// TIA Portal V16 export
// export: Created 2023-06-21T17:06:21.6795389Z, ExportSetting WithDefaults, DisplayName Totally Integrated Automation Portal, DisplayVersion V16 Update 4, DisplayName TIA Portal Version Control Interface, DisplayVersion V16 Update 2, DisplayName TIA Portal Openness, DisplayVersion V16 Update 4, DisplayName SINAMICS Startdrive Advanced, DisplayVersion V16, DisplayName SINAMICS Startdrive G130, G150, S120, S150, SINAMICS MV, S210, DisplayVersion V16, DisplayName SINAMICS Startdrive G110M, G120, G120C, G120D, G120P, DisplayVersion V16, DisplayName STEP 7 Professional, DisplayVersion V16 Update 4, DisplayName STEP 7 Safety, DisplayVersion V16, DisplayName Soft Starter ES, DisplayVersion V16, DisplayName WinCC Advanced, DisplayVersion V16 Update 4
ORGANIZATION_BLOCK "Cyclic interrupt"   // OB30, LAD, CyclicInterrupt
{ S7_Optimized_Access := 'TRUE' }
VERSION : 0.1
// stored: AutoNumber true, IsIECCheckEnabled false, SetENOAutomatically false
   VAR_INPUT
      Initial_Call : Bool;   // Initial call of this OB
      Event_Count : Int;   // Events discarded
   END_VAR
   VAR_TEMP
      Aux_SP_1 : Int;
      Aux_SP_2 : Int;
      Aux_SP_3 : Int;
      Aux_SP_4 : Int;
      Aux_SP_5 : Int;
      Aux_SP_6 : Int;
      Aux_SP_7 : Int;
      Aux_SP_8 : Int;
      Aux_SP_9 : Int;
      Aux_SP_10 : Int;
      Aux_SP_11 : Int;
      Aux_SP_12 : Int;
      Aux_SP_13 : Int;
      Aux_SP_14 : Int;
   END_VAR
   VAR_TEMP   // added for the SCL form of the ladder/FBD networks
      _w1 : Bool;
   END_VAR
BEGIN

REGION Network 2: START
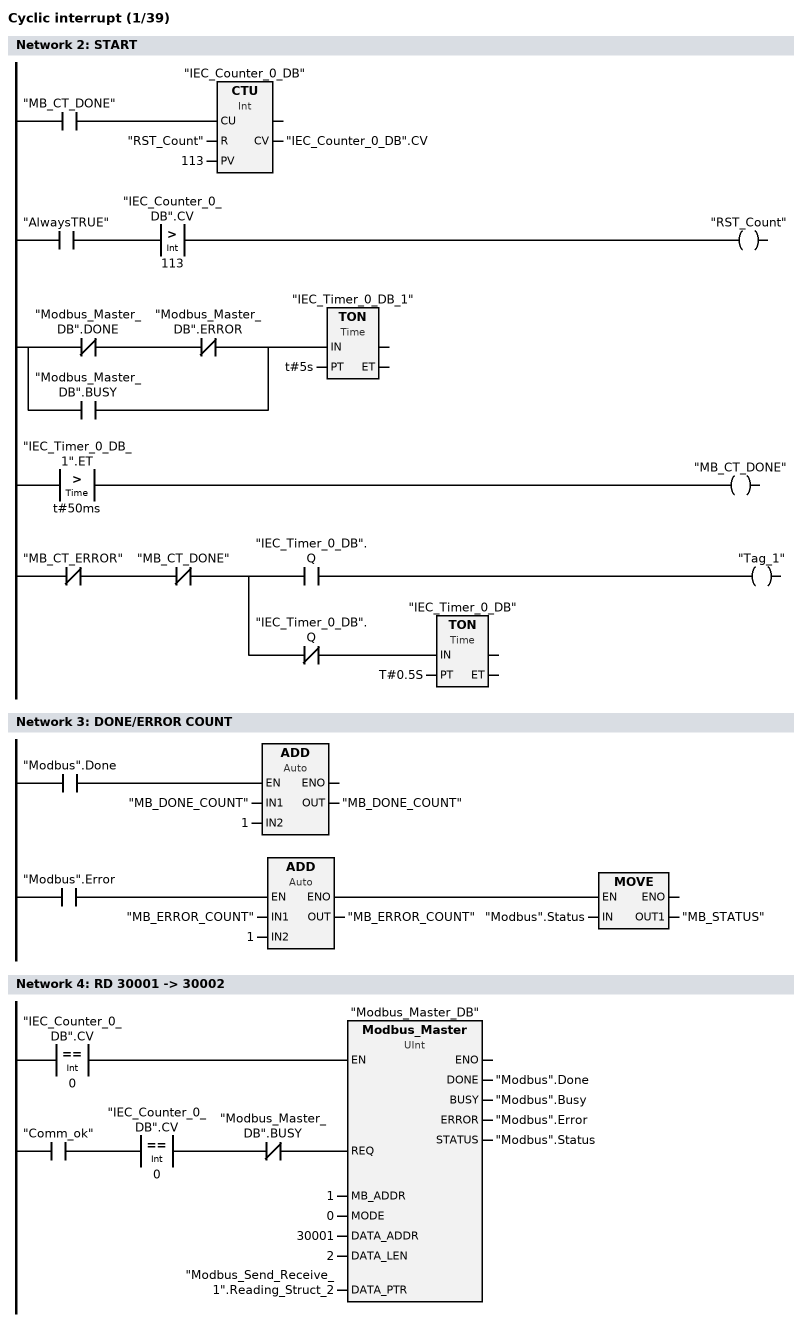
   RUNG wire#powerrail
      Contact( "MB_CT_DONE" )
      { S7_Templates := "value_type := Int" } "IEC_Counter_0_DB".CTU(r := "RST_Count", pv := 113, cv => "IEC_Counter_0_DB".CV)
   END_RUNG
   RUNG wire#powerrail
      Contact( "AlwaysTRUE" )
      { S7_Templates := "SrcType := Int" } GT_Contact(in1 := "IEC_Counter_0_DB".CV, in2 := 113)
      Coil( "RST_Count" )
   END_RUNG
   RUNG wire#powerrail
      I_Contact( "Modbus_Master_DB".DONE )
      I_Contact( "Modbus_Master_DB".ERROR )
      wire#w1
      { S7_Templates := "time_type := Time" } "IEC_Timer_0_DB_1".TON(pt := t#5s, et =>)
   END_RUNG
   RUNG wire#powerrail
      Contact( "Modbus_Master_DB".BUSY )
   END_RUNG wire#w1
   RUNG wire#powerrail
      { S7_Templates := "SrcType := Time" } GT_Contact(in1 := "IEC_Timer_0_DB_1".ET, in2 := t#50ms)
      Coil( "MB_CT_DONE" )
   END_RUNG
   RUNG wire#powerrail
      I_Contact( "MB_CT_ERROR" )
      I_Contact( "MB_CT_DONE" )
      wire#w2
      Contact( "IEC_Timer_0_DB".Q )
      Coil( "Tag_1" )
   END_RUNG
   RUNG wire#w2
      I_Contact( "IEC_Timer_0_DB".Q )
      { S7_Templates := "time_type := Time" } "IEC_Timer_0_DB".TON(pt := T#0.5S, et =>)
   END_RUNG
   // the same network as SCL:
   "IEC_Counter_0_DB".CTU(CU := "MB_CT_DONE", R := "RST_Count", PV := 113, CV => "IEC_Counter_0_DB".CV);
   "RST_Count" := "AlwaysTRUE" AND ("IEC_Counter_0_DB".CV > 113);
   "IEC_Timer_0_DB_1".TON(IN := (NOT "Modbus_Master_DB".DONE AND NOT "Modbus_Master_DB".ERROR) OR "Modbus_Master_DB".BUSY,
                          PT := t#5s);
   "MB_CT_DONE" := "IEC_Timer_0_DB_1".ET > t#50ms;
   #_w1 := NOT "MB_CT_ERROR" AND NOT "MB_CT_DONE";
   "Tag_1" := #_w1 AND "IEC_Timer_0_DB".Q;
   "IEC_Timer_0_DB".TON(IN := #_w1 AND NOT "IEC_Timer_0_DB".Q, PT := T#0.5S);
END_REGION

REGION Network 3: DONE/ERROR COUNT
   RUNG wire#powerrail
      Contact( "Modbus".Done )
      Add(in1 := "MB_DONE_COUNT", in2 := 1, out => "MB_DONE_COUNT")
   END_RUNG
   RUNG wire#powerrail
      Contact( "Modbus".Error )
      Add(in1 := "MB_ERROR_COUNT", in2 := 1, out => "MB_ERROR_COUNT")
      Move(in := "Modbus".Status, out1 => "MB_STATUS")
   END_RUNG
   // the same network as SCL:
   IF "Modbus".Done THEN "MB_DONE_COUNT" := "MB_DONE_COUNT" + 1; END_IF;
   IF "Modbus".Error THEN
       "MB_ERROR_COUNT" := "MB_ERROR_COUNT" + 1;
       "MB_STATUS" := "Modbus".Status;
   END_IF;
END_REGION

REGION Network 4: RD 30001 -> 30002
   RUNG wire#powerrail
      { S7_Templates := "SrcType := Int" } EQ_Contact(in1 := "IEC_Counter_0_DB".CV, in2 := 0)
      { S7_Templates := "[card := 0, word_type := UInt, dword_type := UDInt, byte_type := USInt, any_type := Variant]" } "Modbus_Master_DB".Modbus_Master(REQ := wire#w1, MB_ADDR := 1, MODE := 0, DATA_ADDR := 30001, DATA_LEN := 2, DATA_PTR := "Modbus_Send_Receive_1".Reading_Struct_2, DONE => "Modbus".Done, BUSY => "Modbus".Busy, ERROR => "Modbus".Error, STATUS => "Modbus".Status)
   END_RUNG
   RUNG wire#powerrail
      Contact( "Comm_ok" )
      { S7_Templates := "SrcType := Int" } EQ_Contact(in1 := "IEC_Counter_0_DB".CV, in2 := 0)
      I_Contact( "Modbus_Master_DB".BUSY )
   END_RUNG wire#w1
   // the same network as SCL:
   IF "IEC_Counter_0_DB".CV = 0 THEN
       "Modbus_Master_DB"(REQ := "Comm_ok" AND ("IEC_Counter_0_DB".CV = 0) AND NOT "Modbus_Master_DB".BUSY,   // Modbus_Master
                          MB_ADDR := 1,
                          MODE := 0,
                          DATA_ADDR := 30001,
                          DATA_LEN := 2,
                          DATA_PTR := "Modbus_Send_Receive_1".Reading_Struct_2,
                          DONE => "Modbus".Done,
                          BUSY => "Modbus".Busy,
                          ERROR => "Modbus".Error,
                          STATUS => "Modbus".Status);
   END_IF;
END_REGION

REGION Network 5: STS MAN/AUTO
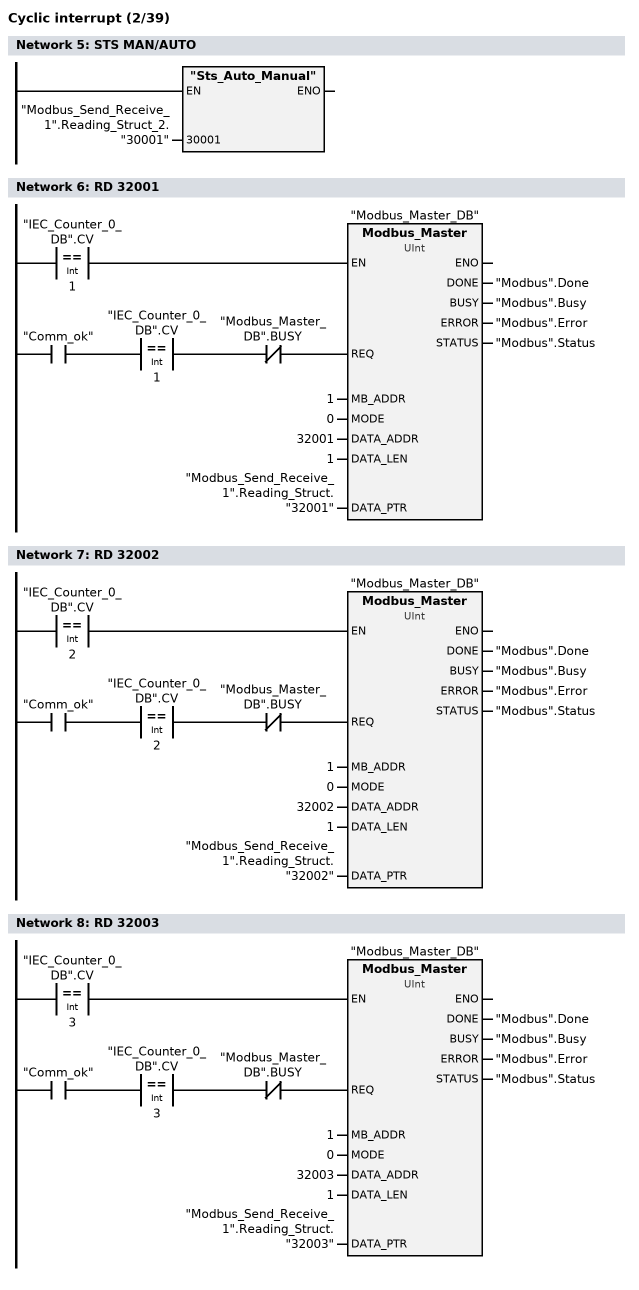
   RUNG wire#powerrail
      "Sts_Auto_Manual"("30001" := "Modbus_Send_Receive_1".Reading_Struct_2."30001")
   END_RUNG
   // the same network as SCL:
   "Sts_Auto_Manual"("30001" := "Modbus_Send_Receive_1".Reading_Struct_2."30001");
END_REGION

REGION Network 6: RD 32001
   RUNG wire#powerrail
      { S7_Templates := "SrcType := Int" } EQ_Contact(in1 := "IEC_Counter_0_DB".CV, in2 := 1)
      { S7_Templates := "[card := 0, word_type := UInt, dword_type := UDInt, byte_type := USInt, any_type := Variant]" } "Modbus_Master_DB".Modbus_Master(REQ := wire#w1, MB_ADDR := 1, MODE := 0, DATA_ADDR := 32001, DATA_LEN := 1, DATA_PTR := "Modbus_Send_Receive_1".Reading_Struct."32001", DONE => "Modbus".Done, BUSY => "Modbus".Busy, ERROR => "Modbus".Error, STATUS => "Modbus".Status)
   END_RUNG
   RUNG wire#powerrail
      Contact( "Comm_ok" )
      { S7_Templates := "SrcType := Int" } EQ_Contact(in1 := "IEC_Counter_0_DB".CV, in2 := 1)
      I_Contact( "Modbus_Master_DB".BUSY )
   END_RUNG wire#w1
   // the same network as SCL:
   IF "IEC_Counter_0_DB".CV = 1 THEN
       "Modbus_Master_DB"(REQ := "Comm_ok" AND ("IEC_Counter_0_DB".CV = 1) AND NOT "Modbus_Master_DB".BUSY,   // Modbus_Master
                          MB_ADDR := 1,
                          MODE := 0,
                          DATA_ADDR := 32001,
                          DATA_LEN := 1,
                          DATA_PTR := "Modbus_Send_Receive_1".Reading_Struct."32001",
                          DONE => "Modbus".Done,
                          BUSY => "Modbus".Busy,
                          ERROR => "Modbus".Error,
                          STATUS => "Modbus".Status);
   END_IF;
END_REGION

REGION Network 7: RD 32002
   RUNG wire#powerrail
      { S7_Templates := "SrcType := Int" } EQ_Contact(in1 := "IEC_Counter_0_DB".CV, in2 := 2)
      { S7_Templates := "[card := 0, word_type := UInt, dword_type := UDInt, byte_type := USInt, any_type := Variant]" } "Modbus_Master_DB".Modbus_Master(REQ := wire#w1, MB_ADDR := 1, MODE := 0, DATA_ADDR := 32002, DATA_LEN := 1, DATA_PTR := "Modbus_Send_Receive_1".Reading_Struct."32002", DONE => "Modbus".Done, BUSY => "Modbus".Busy, ERROR => "Modbus".Error, STATUS => "Modbus".Status)
   END_RUNG
   RUNG wire#powerrail
      Contact( "Comm_ok" )
      { S7_Templates := "SrcType := Int" } EQ_Contact(in1 := "IEC_Counter_0_DB".CV, in2 := 2)
      I_Contact( "Modbus_Master_DB".BUSY )
   END_RUNG wire#w1
   // the same network as SCL:
   IF "IEC_Counter_0_DB".CV = 2 THEN
       "Modbus_Master_DB"(REQ := "Comm_ok" AND ("IEC_Counter_0_DB".CV = 2) AND NOT "Modbus_Master_DB".BUSY,   // Modbus_Master
                          MB_ADDR := 1,
                          MODE := 0,
                          DATA_ADDR := 32002,
                          DATA_LEN := 1,
                          DATA_PTR := "Modbus_Send_Receive_1".Reading_Struct."32002",
                          DONE => "Modbus".Done,
                          BUSY => "Modbus".Busy,
                          ERROR => "Modbus".Error,
                          STATUS => "Modbus".Status);
   END_IF;
END_REGION

REGION Network 8: RD 32003
   RUNG wire#powerrail
      { S7_Templates := "SrcType := Int" } EQ_Contact(in1 := "IEC_Counter_0_DB".CV, in2 := 3)
      { S7_Templates := "[card := 0, word_type := UInt, dword_type := UDInt, byte_type := USInt, any_type := Variant]" } "Modbus_Master_DB".Modbus_Master(REQ := wire#w1, MB_ADDR := 1, MODE := 0, DATA_ADDR := 32003, DATA_LEN := 1, DATA_PTR := "Modbus_Send_Receive_1".Reading_Struct."32003", DONE => "Modbus".Done, BUSY => "Modbus".Busy, ERROR => "Modbus".Error, STATUS => "Modbus".Status)
   END_RUNG
   RUNG wire#powerrail
      Contact( "Comm_ok" )
      { S7_Templates := "SrcType := Int" } EQ_Contact(in1 := "IEC_Counter_0_DB".CV, in2 := 3)
      I_Contact( "Modbus_Master_DB".BUSY )
   END_RUNG wire#w1
   // the same network as SCL:
   IF "IEC_Counter_0_DB".CV = 3 THEN
       "Modbus_Master_DB"(REQ := "Comm_ok" AND ("IEC_Counter_0_DB".CV = 3) AND NOT "Modbus_Master_DB".BUSY,   // Modbus_Master
                          MB_ADDR := 1,
                          MODE := 0,
                          DATA_ADDR := 32003,
                          DATA_LEN := 1,
                          DATA_PTR := "Modbus_Send_Receive_1".Reading_Struct."32003",
                          DONE => "Modbus".Done,
                          BUSY => "Modbus".Busy,
                          ERROR => "Modbus".Error,
                          STATUS => "Modbus".Status);
   END_IF;
END_REGION

REGION Network 9: RD 32004
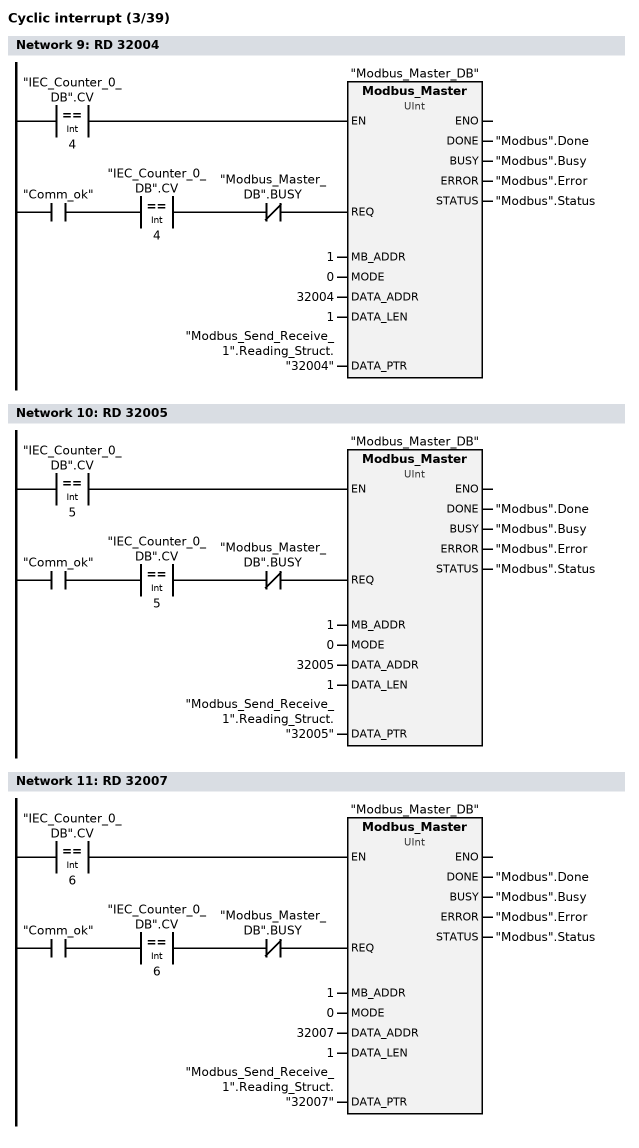
   RUNG wire#powerrail
      { S7_Templates := "SrcType := Int" } EQ_Contact(in1 := "IEC_Counter_0_DB".CV, in2 := 4)
      { S7_Templates := "[card := 0, word_type := UInt, dword_type := UDInt, byte_type := USInt, any_type := Variant]" } "Modbus_Master_DB".Modbus_Master(REQ := wire#w1, MB_ADDR := 1, MODE := 0, DATA_ADDR := 32004, DATA_LEN := 1, DATA_PTR := "Modbus_Send_Receive_1".Reading_Struct."32004", DONE => "Modbus".Done, BUSY => "Modbus".Busy, ERROR => "Modbus".Error, STATUS => "Modbus".Status)
   END_RUNG
   RUNG wire#powerrail
      Contact( "Comm_ok" )
      { S7_Templates := "SrcType := Int" } EQ_Contact(in1 := "IEC_Counter_0_DB".CV, in2 := 4)
      I_Contact( "Modbus_Master_DB".BUSY )
   END_RUNG wire#w1
   // the same network as SCL:
   IF "IEC_Counter_0_DB".CV = 4 THEN
       "Modbus_Master_DB"(REQ := "Comm_ok" AND ("IEC_Counter_0_DB".CV = 4) AND NOT "Modbus_Master_DB".BUSY,   // Modbus_Master
                          MB_ADDR := 1,
                          MODE := 0,
                          DATA_ADDR := 32004,
                          DATA_LEN := 1,
                          DATA_PTR := "Modbus_Send_Receive_1".Reading_Struct."32004",
                          DONE => "Modbus".Done,
                          BUSY => "Modbus".Busy,
                          ERROR => "Modbus".Error,
                          STATUS => "Modbus".Status);
   END_IF;
END_REGION

REGION Network 10: RD 32005
   RUNG wire#powerrail
      { S7_Templates := "SrcType := Int" } EQ_Contact(in1 := "IEC_Counter_0_DB".CV, in2 := 5)
      { S7_Templates := "[card := 0, word_type := UInt, dword_type := UDInt, byte_type := USInt, any_type := Variant]" } "Modbus_Master_DB".Modbus_Master(REQ := wire#w1, MB_ADDR := 1, MODE := 0, DATA_ADDR := 32005, DATA_LEN := 1, DATA_PTR := "Modbus_Send_Receive_1".Reading_Struct."32005", DONE => "Modbus".Done, BUSY => "Modbus".Busy, ERROR => "Modbus".Error, STATUS => "Modbus".Status)
   END_RUNG
   RUNG wire#powerrail
      Contact( "Comm_ok" )
      { S7_Templates := "SrcType := Int" } EQ_Contact(in1 := "IEC_Counter_0_DB".CV, in2 := 5)
      I_Contact( "Modbus_Master_DB".BUSY )
   END_RUNG wire#w1
   // the same network as SCL:
   IF "IEC_Counter_0_DB".CV = 5 THEN
       "Modbus_Master_DB"(REQ := "Comm_ok" AND ("IEC_Counter_0_DB".CV = 5) AND NOT "Modbus_Master_DB".BUSY,   // Modbus_Master
                          MB_ADDR := 1,
                          MODE := 0,
                          DATA_ADDR := 32005,
                          DATA_LEN := 1,
                          DATA_PTR := "Modbus_Send_Receive_1".Reading_Struct."32005",
                          DONE => "Modbus".Done,
                          BUSY => "Modbus".Busy,
                          ERROR => "Modbus".Error,
                          STATUS => "Modbus".Status);
   END_IF;
END_REGION

REGION Network 11: RD 32007
   RUNG wire#powerrail
      { S7_Templates := "SrcType := Int" } EQ_Contact(in1 := "IEC_Counter_0_DB".CV, in2 := 6)
      { S7_Templates := "[card := 0, word_type := UInt, dword_type := UDInt, byte_type := USInt, any_type := Variant]" } "Modbus_Master_DB".Modbus_Master(REQ := wire#w1, MB_ADDR := 1, MODE := 0, DATA_ADDR := 32007, DATA_LEN := 1, DATA_PTR := "Modbus_Send_Receive_1".Reading_Struct."32007", DONE => "Modbus".Done, BUSY => "Modbus".Busy, ERROR => "Modbus".Error, STATUS => "Modbus".Status)
   END_RUNG
   RUNG wire#powerrail
      Contact( "Comm_ok" )
      { S7_Templates := "SrcType := Int" } EQ_Contact(in1 := "IEC_Counter_0_DB".CV, in2 := 6)
      I_Contact( "Modbus_Master_DB".BUSY )
   END_RUNG wire#w1
   // the same network as SCL:
   IF "IEC_Counter_0_DB".CV = 6 THEN
       "Modbus_Master_DB"(REQ := "Comm_ok" AND ("IEC_Counter_0_DB".CV = 6) AND NOT "Modbus_Master_DB".BUSY,   // Modbus_Master
                          MB_ADDR := 1,
                          MODE := 0,
                          DATA_ADDR := 32007,
                          DATA_LEN := 1,
                          DATA_PTR := "Modbus_Send_Receive_1".Reading_Struct."32007",
                          DONE => "Modbus".Done,
                          BUSY => "Modbus".Busy,
                          ERROR => "Modbus".Error,
                          STATUS => "Modbus".Status);
   END_IF;
END_REGION

REGION Network 12: RD 32008
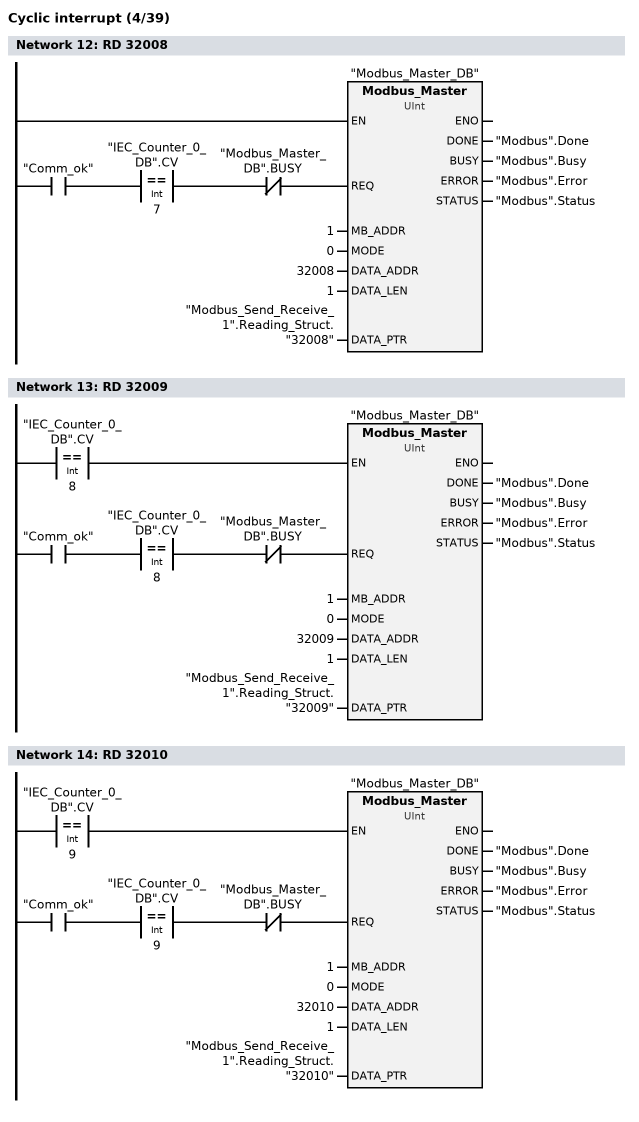
   RUNG wire#powerrail
      { S7_Templates := "[card := 0, word_type := UInt, dword_type := UDInt, byte_type := USInt, any_type := Variant]" } "Modbus_Master_DB".Modbus_Master(REQ := wire#w1, MB_ADDR := 1, MODE := 0, DATA_ADDR := 32008, DATA_LEN := 1, DATA_PTR := "Modbus_Send_Receive_1".Reading_Struct."32008", DONE => "Modbus".Done, BUSY => "Modbus".Busy, ERROR => "Modbus".Error, STATUS => "Modbus".Status)
   END_RUNG
   RUNG wire#powerrail
      Contact( "Comm_ok" )
      { S7_Templates := "SrcType := Int" } EQ_Contact(in1 := "IEC_Counter_0_DB".CV, in2 := 7)
      I_Contact( "Modbus_Master_DB".BUSY )
   END_RUNG wire#w1
   // the same network as SCL:
   "Modbus_Master_DB"(REQ := "Comm_ok" AND ("IEC_Counter_0_DB".CV = 7) AND NOT "Modbus_Master_DB".BUSY,   // Modbus_Master
                      MB_ADDR := 1,
                      MODE := 0,
                      DATA_ADDR := 32008,
                      DATA_LEN := 1,
                      DATA_PTR := "Modbus_Send_Receive_1".Reading_Struct."32008",
                      DONE => "Modbus".Done,
                      BUSY => "Modbus".Busy,
                      ERROR => "Modbus".Error,
                      STATUS => "Modbus".Status);
END_REGION

REGION Network 13: RD 32009
   RUNG wire#powerrail
      { S7_Templates := "SrcType := Int" } EQ_Contact(in1 := "IEC_Counter_0_DB".CV, in2 := 8)
      { S7_Templates := "[card := 0, word_type := UInt, dword_type := UDInt, byte_type := USInt, any_type := Variant]" } "Modbus_Master_DB".Modbus_Master(REQ := wire#w1, MB_ADDR := 1, MODE := 0, DATA_ADDR := 32009, DATA_LEN := 1, DATA_PTR := "Modbus_Send_Receive_1".Reading_Struct."32009", DONE => "Modbus".Done, BUSY => "Modbus".Busy, ERROR => "Modbus".Error, STATUS => "Modbus".Status)
   END_RUNG
   RUNG wire#powerrail
      Contact( "Comm_ok" )
      { S7_Templates := "SrcType := Int" } EQ_Contact(in1 := "IEC_Counter_0_DB".CV, in2 := 8)
      I_Contact( "Modbus_Master_DB".BUSY )
   END_RUNG wire#w1
   // the same network as SCL:
   IF "IEC_Counter_0_DB".CV = 8 THEN
       "Modbus_Master_DB"(REQ := "Comm_ok" AND ("IEC_Counter_0_DB".CV = 8) AND NOT "Modbus_Master_DB".BUSY,   // Modbus_Master
                          MB_ADDR := 1,
                          MODE := 0,
                          DATA_ADDR := 32009,
                          DATA_LEN := 1,
                          DATA_PTR := "Modbus_Send_Receive_1".Reading_Struct."32009",
                          DONE => "Modbus".Done,
                          BUSY => "Modbus".Busy,
                          ERROR => "Modbus".Error,
                          STATUS => "Modbus".Status);
   END_IF;
END_REGION

REGION Network 14: RD 32010
   RUNG wire#powerrail
      { S7_Templates := "SrcType := Int" } EQ_Contact(in1 := "IEC_Counter_0_DB".CV, in2 := 9)
      { S7_Templates := "[card := 0, word_type := UInt, dword_type := UDInt, byte_type := USInt, any_type := Variant]" } "Modbus_Master_DB".Modbus_Master(REQ := wire#w1, MB_ADDR := 1, MODE := 0, DATA_ADDR := 32010, DATA_LEN := 1, DATA_PTR := "Modbus_Send_Receive_1".Reading_Struct."32010", DONE => "Modbus".Done, BUSY => "Modbus".Busy, ERROR => "Modbus".Error, STATUS => "Modbus".Status)
   END_RUNG
   RUNG wire#powerrail
      Contact( "Comm_ok" )
      { S7_Templates := "SrcType := Int" } EQ_Contact(in1 := "IEC_Counter_0_DB".CV, in2 := 9)
      I_Contact( "Modbus_Master_DB".BUSY )
   END_RUNG wire#w1
   // the same network as SCL:
   IF "IEC_Counter_0_DB".CV = 9 THEN
       "Modbus_Master_DB"(REQ := "Comm_ok" AND ("IEC_Counter_0_DB".CV = 9) AND NOT "Modbus_Master_DB".BUSY,   // Modbus_Master
                          MB_ADDR := 1,
                          MODE := 0,
                          DATA_ADDR := 32010,
                          DATA_LEN := 1,
                          DATA_PTR := "Modbus_Send_Receive_1".Reading_Struct."32010",
                          DONE => "Modbus".Done,
                          BUSY => "Modbus".Busy,
                          ERROR => "Modbus".Error,
                          STATUS => "Modbus".Status);
   END_IF;
END_REGION

REGION Network 15: RD 32011
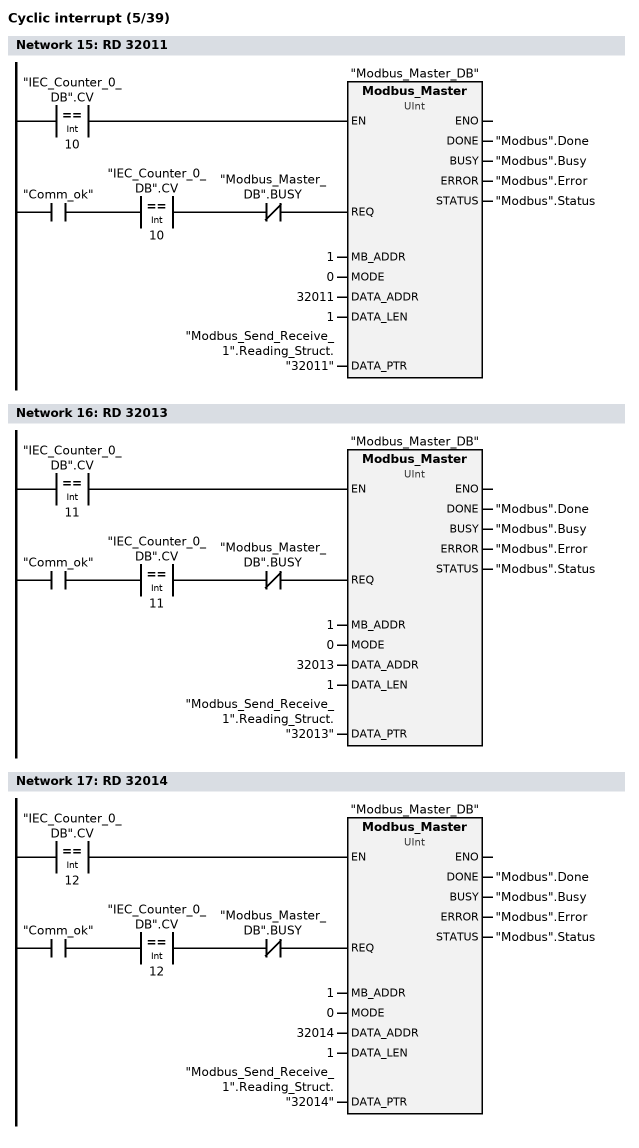
   RUNG wire#powerrail
      { S7_Templates := "SrcType := Int" } EQ_Contact(in1 := "IEC_Counter_0_DB".CV, in2 := 10)
      { S7_Templates := "[card := 0, word_type := UInt, dword_type := UDInt, byte_type := USInt, any_type := Variant]" } "Modbus_Master_DB".Modbus_Master(REQ := wire#w1, MB_ADDR := 1, MODE := 0, DATA_ADDR := 32011, DATA_LEN := 1, DATA_PTR := "Modbus_Send_Receive_1".Reading_Struct."32011", DONE => "Modbus".Done, BUSY => "Modbus".Busy, ERROR => "Modbus".Error, STATUS => "Modbus".Status)
   END_RUNG
   RUNG wire#powerrail
      Contact( "Comm_ok" )
      { S7_Templates := "SrcType := Int" } EQ_Contact(in1 := "IEC_Counter_0_DB".CV, in2 := 10)
      I_Contact( "Modbus_Master_DB".BUSY )
   END_RUNG wire#w1
   // the same network as SCL:
   IF "IEC_Counter_0_DB".CV = 10 THEN
       "Modbus_Master_DB"(REQ := "Comm_ok" AND ("IEC_Counter_0_DB".CV = 10) AND NOT "Modbus_Master_DB".BUSY,   // Modbus_Master
                          MB_ADDR := 1,
                          MODE := 0,
                          DATA_ADDR := 32011,
                          DATA_LEN := 1,
                          DATA_PTR := "Modbus_Send_Receive_1".Reading_Struct."32011",
                          DONE => "Modbus".Done,
                          BUSY => "Modbus".Busy,
                          ERROR => "Modbus".Error,
                          STATUS => "Modbus".Status);
   END_IF;
END_REGION

REGION Network 16: RD 32013
   RUNG wire#powerrail
      { S7_Templates := "SrcType := Int" } EQ_Contact(in1 := "IEC_Counter_0_DB".CV, in2 := 11)
      { S7_Templates := "[card := 0, word_type := UInt, dword_type := UDInt, byte_type := USInt, any_type := Variant]" } "Modbus_Master_DB".Modbus_Master(REQ := wire#w1, MB_ADDR := 1, MODE := 0, DATA_ADDR := 32013, DATA_LEN := 1, DATA_PTR := "Modbus_Send_Receive_1".Reading_Struct."32013", DONE => "Modbus".Done, BUSY => "Modbus".Busy, ERROR => "Modbus".Error, STATUS => "Modbus".Status)
   END_RUNG
   RUNG wire#powerrail
      Contact( "Comm_ok" )
      { S7_Templates := "SrcType := Int" } EQ_Contact(in1 := "IEC_Counter_0_DB".CV, in2 := 11)
      I_Contact( "Modbus_Master_DB".BUSY )
   END_RUNG wire#w1
   // the same network as SCL:
   IF "IEC_Counter_0_DB".CV = 11 THEN
       "Modbus_Master_DB"(REQ := "Comm_ok" AND ("IEC_Counter_0_DB".CV = 11) AND NOT "Modbus_Master_DB".BUSY,   // Modbus_Master
                          MB_ADDR := 1,
                          MODE := 0,
                          DATA_ADDR := 32013,
                          DATA_LEN := 1,
                          DATA_PTR := "Modbus_Send_Receive_1".Reading_Struct."32013",
                          DONE => "Modbus".Done,
                          BUSY => "Modbus".Busy,
                          ERROR => "Modbus".Error,
                          STATUS => "Modbus".Status);
   END_IF;
END_REGION

REGION Network 17: RD 32014
   RUNG wire#powerrail
      { S7_Templates := "SrcType := Int" } EQ_Contact(in1 := "IEC_Counter_0_DB".CV, in2 := 12)
      { S7_Templates := "[card := 0, word_type := UInt, dword_type := UDInt, byte_type := USInt, any_type := Variant]" } "Modbus_Master_DB".Modbus_Master(REQ := wire#w1, MB_ADDR := 1, MODE := 0, DATA_ADDR := 32014, DATA_LEN := 1, DATA_PTR := "Modbus_Send_Receive_1".Reading_Struct."32014", DONE => "Modbus".Done, BUSY => "Modbus".Busy, ERROR => "Modbus".Error, STATUS => "Modbus".Status)
   END_RUNG
   RUNG wire#powerrail
      Contact( "Comm_ok" )
      { S7_Templates := "SrcType := Int" } EQ_Contact(in1 := "IEC_Counter_0_DB".CV, in2 := 12)
      I_Contact( "Modbus_Master_DB".BUSY )
   END_RUNG wire#w1
   // the same network as SCL:
   IF "IEC_Counter_0_DB".CV = 12 THEN
       "Modbus_Master_DB"(REQ := "Comm_ok" AND ("IEC_Counter_0_DB".CV = 12) AND NOT "Modbus_Master_DB".BUSY,   // Modbus_Master
                          MB_ADDR := 1,
                          MODE := 0,
                          DATA_ADDR := 32014,
                          DATA_LEN := 1,
                          DATA_PTR := "Modbus_Send_Receive_1".Reading_Struct."32014",
                          DONE => "Modbus".Done,
                          BUSY => "Modbus".Busy,
                          ERROR => "Modbus".Error,
                          STATUS => "Modbus".Status);
   END_IF;
END_REGION

REGION Network 18: RD 32015
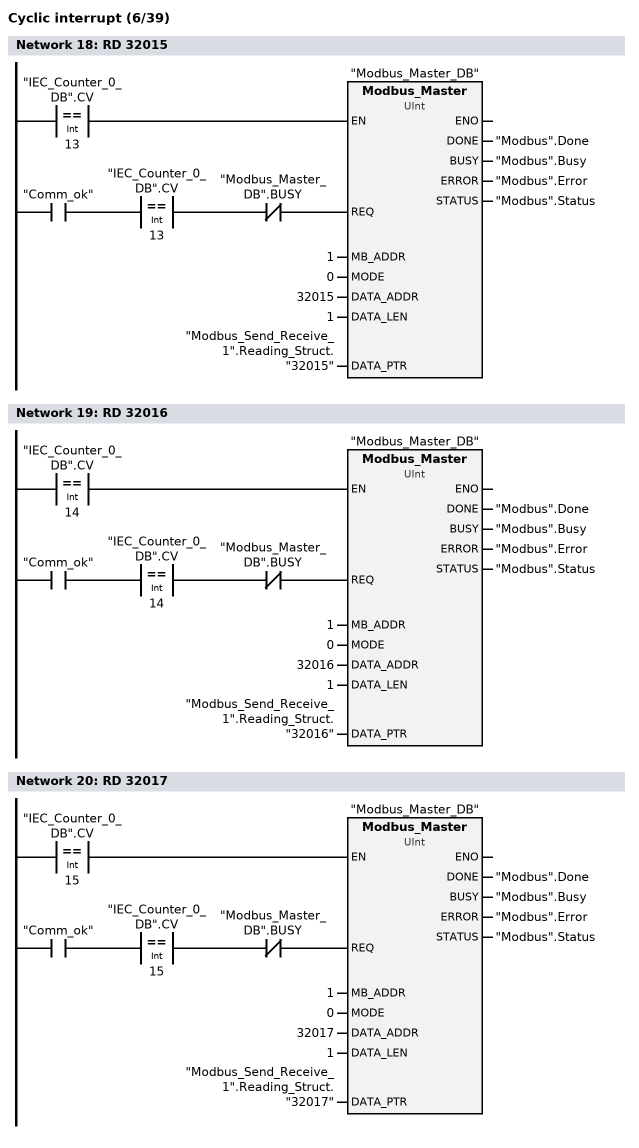
   RUNG wire#powerrail
      { S7_Templates := "SrcType := Int" } EQ_Contact(in1 := "IEC_Counter_0_DB".CV, in2 := 13)
      { S7_Templates := "[card := 0, word_type := UInt, dword_type := UDInt, byte_type := USInt, any_type := Variant]" } "Modbus_Master_DB".Modbus_Master(REQ := wire#w1, MB_ADDR := 1, MODE := 0, DATA_ADDR := 32015, DATA_LEN := 1, DATA_PTR := "Modbus_Send_Receive_1".Reading_Struct."32015", DONE => "Modbus".Done, BUSY => "Modbus".Busy, ERROR => "Modbus".Error, STATUS => "Modbus".Status)
   END_RUNG
   RUNG wire#powerrail
      Contact( "Comm_ok" )
      { S7_Templates := "SrcType := Int" } EQ_Contact(in1 := "IEC_Counter_0_DB".CV, in2 := 13)
      I_Contact( "Modbus_Master_DB".BUSY )
   END_RUNG wire#w1
   // the same network as SCL:
   IF "IEC_Counter_0_DB".CV = 13 THEN
       "Modbus_Master_DB"(REQ := "Comm_ok" AND ("IEC_Counter_0_DB".CV = 13) AND NOT "Modbus_Master_DB".BUSY,   // Modbus_Master
                          MB_ADDR := 1,
                          MODE := 0,
                          DATA_ADDR := 32015,
                          DATA_LEN := 1,
                          DATA_PTR := "Modbus_Send_Receive_1".Reading_Struct."32015",
                          DONE => "Modbus".Done,
                          BUSY => "Modbus".Busy,
                          ERROR => "Modbus".Error,
                          STATUS => "Modbus".Status);
   END_IF;
END_REGION

REGION Network 19: RD 32016
   RUNG wire#powerrail
      { S7_Templates := "SrcType := Int" } EQ_Contact(in1 := "IEC_Counter_0_DB".CV, in2 := 14)
      { S7_Templates := "[card := 0, word_type := UInt, dword_type := UDInt, byte_type := USInt, any_type := Variant]" } "Modbus_Master_DB".Modbus_Master(REQ := wire#w1, MB_ADDR := 1, MODE := 0, DATA_ADDR := 32016, DATA_LEN := 1, DATA_PTR := "Modbus_Send_Receive_1".Reading_Struct."32016", DONE => "Modbus".Done, BUSY => "Modbus".Busy, ERROR => "Modbus".Error, STATUS => "Modbus".Status)
   END_RUNG
   RUNG wire#powerrail
      Contact( "Comm_ok" )
      { S7_Templates := "SrcType := Int" } EQ_Contact(in1 := "IEC_Counter_0_DB".CV, in2 := 14)
      I_Contact( "Modbus_Master_DB".BUSY )
   END_RUNG wire#w1
   // the same network as SCL:
   IF "IEC_Counter_0_DB".CV = 14 THEN
       "Modbus_Master_DB"(REQ := "Comm_ok" AND ("IEC_Counter_0_DB".CV = 14) AND NOT "Modbus_Master_DB".BUSY,   // Modbus_Master
                          MB_ADDR := 1,
                          MODE := 0,
                          DATA_ADDR := 32016,
                          DATA_LEN := 1,
                          DATA_PTR := "Modbus_Send_Receive_1".Reading_Struct."32016",
                          DONE => "Modbus".Done,
                          BUSY => "Modbus".Busy,
                          ERROR => "Modbus".Error,
                          STATUS => "Modbus".Status);
   END_IF;
END_REGION

REGION Network 20: RD 32017
   RUNG wire#powerrail
      { S7_Templates := "SrcType := Int" } EQ_Contact(in1 := "IEC_Counter_0_DB".CV, in2 := 15)
      { S7_Templates := "[card := 0, word_type := UInt, dword_type := UDInt, byte_type := USInt, any_type := Variant]" } "Modbus_Master_DB".Modbus_Master(REQ := wire#w1, MB_ADDR := 1, MODE := 0, DATA_ADDR := 32017, DATA_LEN := 1, DATA_PTR := "Modbus_Send_Receive_1".Reading_Struct."32017", DONE => "Modbus".Done, BUSY => "Modbus".Busy, ERROR => "Modbus".Error, STATUS => "Modbus".Status)
   END_RUNG
   RUNG wire#powerrail
      Contact( "Comm_ok" )
      { S7_Templates := "SrcType := Int" } EQ_Contact(in1 := "IEC_Counter_0_DB".CV, in2 := 15)
      I_Contact( "Modbus_Master_DB".BUSY )
   END_RUNG wire#w1
   // the same network as SCL:
   IF "IEC_Counter_0_DB".CV = 15 THEN
       "Modbus_Master_DB"(REQ := "Comm_ok" AND ("IEC_Counter_0_DB".CV = 15) AND NOT "Modbus_Master_DB".BUSY,   // Modbus_Master
                          MB_ADDR := 1,
                          MODE := 0,
                          DATA_ADDR := 32017,
                          DATA_LEN := 1,
                          DATA_PTR := "Modbus_Send_Receive_1".Reading_Struct."32017",
                          DONE => "Modbus".Done,
                          BUSY => "Modbus".Busy,
                          ERROR => "Modbus".Error,
                          STATUS => "Modbus".Status);
   END_IF;
END_REGION

REGION Network 21: RD 32019
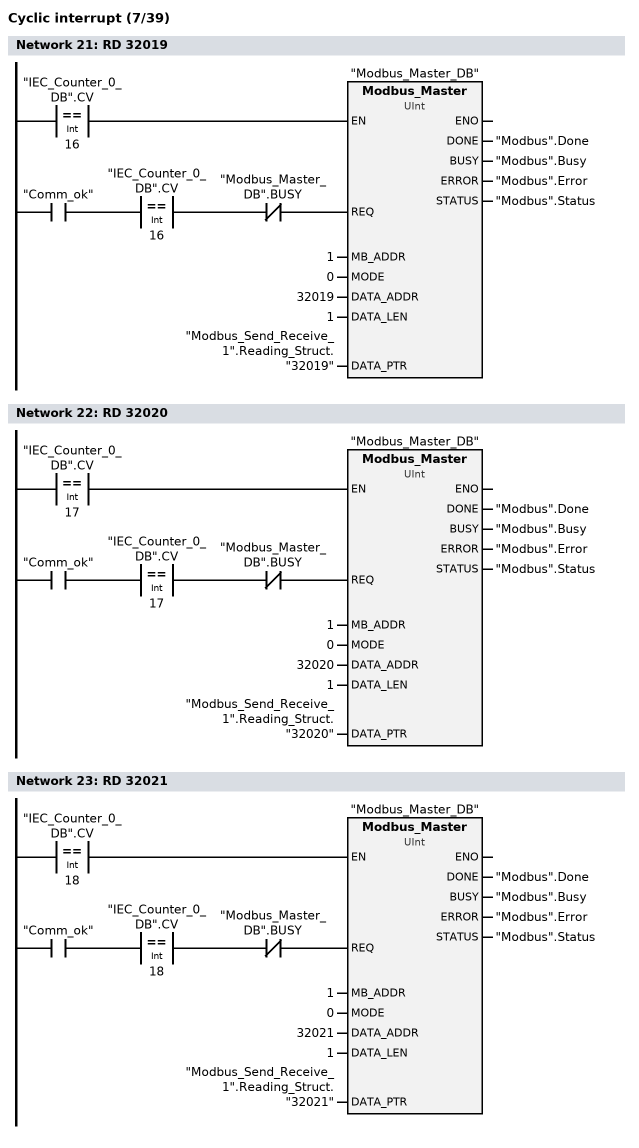
   RUNG wire#powerrail
      { S7_Templates := "SrcType := Int" } EQ_Contact(in1 := "IEC_Counter_0_DB".CV, in2 := 16)
      { S7_Templates := "[card := 0, word_type := UInt, dword_type := UDInt, byte_type := USInt, any_type := Variant]" } "Modbus_Master_DB".Modbus_Master(REQ := wire#w1, MB_ADDR := 1, MODE := 0, DATA_ADDR := 32019, DATA_LEN := 1, DATA_PTR := "Modbus_Send_Receive_1".Reading_Struct."32019", DONE => "Modbus".Done, BUSY => "Modbus".Busy, ERROR => "Modbus".Error, STATUS => "Modbus".Status)
   END_RUNG
   RUNG wire#powerrail
      Contact( "Comm_ok" )
      { S7_Templates := "SrcType := Int" } EQ_Contact(in1 := "IEC_Counter_0_DB".CV, in2 := 16)
      I_Contact( "Modbus_Master_DB".BUSY )
   END_RUNG wire#w1
   // the same network as SCL:
   IF "IEC_Counter_0_DB".CV = 16 THEN
       "Modbus_Master_DB"(REQ := "Comm_ok" AND ("IEC_Counter_0_DB".CV = 16) AND NOT "Modbus_Master_DB".BUSY,   // Modbus_Master
                          MB_ADDR := 1,
                          MODE := 0,
                          DATA_ADDR := 32019,
                          DATA_LEN := 1,
                          DATA_PTR := "Modbus_Send_Receive_1".Reading_Struct."32019",
                          DONE => "Modbus".Done,
                          BUSY => "Modbus".Busy,
                          ERROR => "Modbus".Error,
                          STATUS => "Modbus".Status);
   END_IF;
END_REGION

REGION Network 22: RD 32020
   RUNG wire#powerrail
      { S7_Templates := "SrcType := Int" } EQ_Contact(in1 := "IEC_Counter_0_DB".CV, in2 := 17)
      { S7_Templates := "[card := 0, word_type := UInt, dword_type := UDInt, byte_type := USInt, any_type := Variant]" } "Modbus_Master_DB".Modbus_Master(REQ := wire#w1, MB_ADDR := 1, MODE := 0, DATA_ADDR := 32020, DATA_LEN := 1, DATA_PTR := "Modbus_Send_Receive_1".Reading_Struct."32020", DONE => "Modbus".Done, BUSY => "Modbus".Busy, ERROR => "Modbus".Error, STATUS => "Modbus".Status)
   END_RUNG
   RUNG wire#powerrail
      Contact( "Comm_ok" )
      { S7_Templates := "SrcType := Int" } EQ_Contact(in1 := "IEC_Counter_0_DB".CV, in2 := 17)
      I_Contact( "Modbus_Master_DB".BUSY )
   END_RUNG wire#w1
   // the same network as SCL:
   IF "IEC_Counter_0_DB".CV = 17 THEN
       "Modbus_Master_DB"(REQ := "Comm_ok" AND ("IEC_Counter_0_DB".CV = 17) AND NOT "Modbus_Master_DB".BUSY,   // Modbus_Master
                          MB_ADDR := 1,
                          MODE := 0,
                          DATA_ADDR := 32020,
                          DATA_LEN := 1,
                          DATA_PTR := "Modbus_Send_Receive_1".Reading_Struct."32020",
                          DONE => "Modbus".Done,
                          BUSY => "Modbus".Busy,
                          ERROR => "Modbus".Error,
                          STATUS => "Modbus".Status);
   END_IF;
END_REGION

REGION Network 23: RD 32021
   RUNG wire#powerrail
      { S7_Templates := "SrcType := Int" } EQ_Contact(in1 := "IEC_Counter_0_DB".CV, in2 := 18)
      { S7_Templates := "[card := 0, word_type := UInt, dword_type := UDInt, byte_type := USInt, any_type := Variant]" } "Modbus_Master_DB".Modbus_Master(REQ := wire#w1, MB_ADDR := 1, MODE := 0, DATA_ADDR := 32021, DATA_LEN := 1, DATA_PTR := "Modbus_Send_Receive_1".Reading_Struct."32021", DONE => "Modbus".Done, BUSY => "Modbus".Busy, ERROR => "Modbus".Error, STATUS => "Modbus".Status)
   END_RUNG
   RUNG wire#powerrail
      Contact( "Comm_ok" )
      { S7_Templates := "SrcType := Int" } EQ_Contact(in1 := "IEC_Counter_0_DB".CV, in2 := 18)
      I_Contact( "Modbus_Master_DB".BUSY )
   END_RUNG wire#w1
   // the same network as SCL:
   IF "IEC_Counter_0_DB".CV = 18 THEN
       "Modbus_Master_DB"(REQ := "Comm_ok" AND ("IEC_Counter_0_DB".CV = 18) AND NOT "Modbus_Master_DB".BUSY,   // Modbus_Master
                          MB_ADDR := 1,
                          MODE := 0,
                          DATA_ADDR := 32021,
                          DATA_LEN := 1,
                          DATA_PTR := "Modbus_Send_Receive_1".Reading_Struct."32021",
                          DONE => "Modbus".Done,
                          BUSY => "Modbus".Busy,
                          ERROR => "Modbus".Error,
                          STATUS => "Modbus".Status);
   END_IF;
END_REGION

REGION Network 24: RD 32022
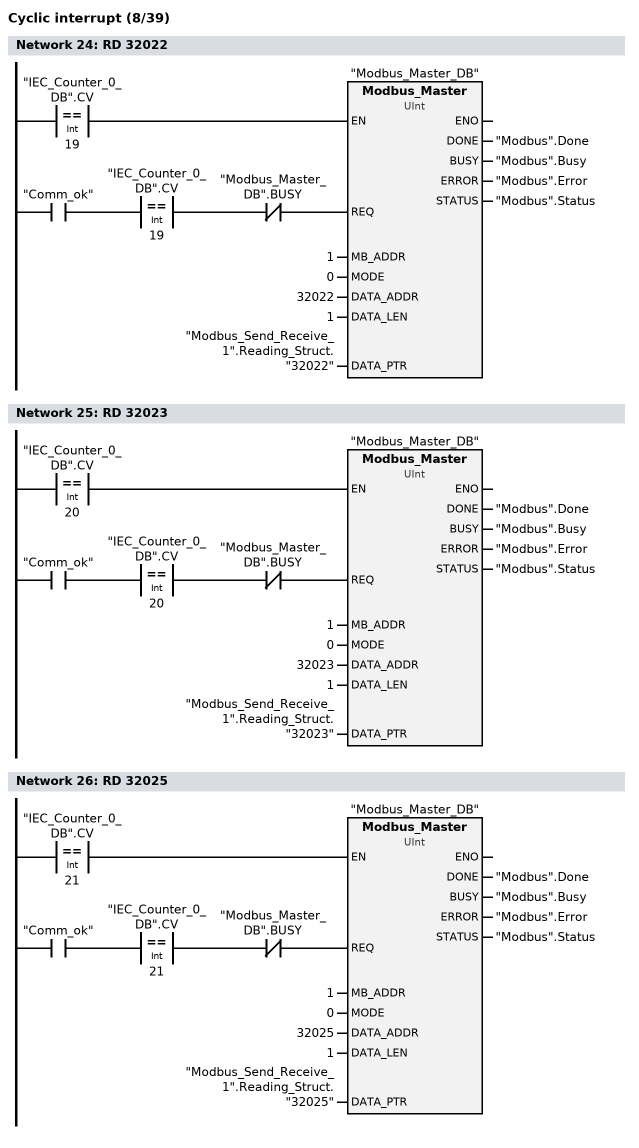
   RUNG wire#powerrail
      { S7_Templates := "SrcType := Int" } EQ_Contact(in1 := "IEC_Counter_0_DB".CV, in2 := 19)
      { S7_Templates := "[card := 0, word_type := UInt, dword_type := UDInt, byte_type := USInt, any_type := Variant]" } "Modbus_Master_DB".Modbus_Master(REQ := wire#w1, MB_ADDR := 1, MODE := 0, DATA_ADDR := 32022, DATA_LEN := 1, DATA_PTR := "Modbus_Send_Receive_1".Reading_Struct."32022", DONE => "Modbus".Done, BUSY => "Modbus".Busy, ERROR => "Modbus".Error, STATUS => "Modbus".Status)
   END_RUNG
   RUNG wire#powerrail
      Contact( "Comm_ok" )
      { S7_Templates := "SrcType := Int" } EQ_Contact(in1 := "IEC_Counter_0_DB".CV, in2 := 19)
      I_Contact( "Modbus_Master_DB".BUSY )
   END_RUNG wire#w1
   // the same network as SCL:
   IF "IEC_Counter_0_DB".CV = 19 THEN
       "Modbus_Master_DB"(REQ := "Comm_ok" AND ("IEC_Counter_0_DB".CV = 19) AND NOT "Modbus_Master_DB".BUSY,   // Modbus_Master
                          MB_ADDR := 1,
                          MODE := 0,
                          DATA_ADDR := 32022,
                          DATA_LEN := 1,
                          DATA_PTR := "Modbus_Send_Receive_1".Reading_Struct."32022",
                          DONE => "Modbus".Done,
                          BUSY => "Modbus".Busy,
                          ERROR => "Modbus".Error,
                          STATUS => "Modbus".Status);
   END_IF;
END_REGION

REGION Network 25: RD 32023
   RUNG wire#powerrail
      { S7_Templates := "SrcType := Int" } EQ_Contact(in1 := "IEC_Counter_0_DB".CV, in2 := 20)
      { S7_Templates := "[card := 0, word_type := UInt, dword_type := UDInt, byte_type := USInt, any_type := Variant]" } "Modbus_Master_DB".Modbus_Master(REQ := wire#w1, MB_ADDR := 1, MODE := 0, DATA_ADDR := 32023, DATA_LEN := 1, DATA_PTR := "Modbus_Send_Receive_1".Reading_Struct."32023", DONE => "Modbus".Done, BUSY => "Modbus".Busy, ERROR => "Modbus".Error, STATUS => "Modbus".Status)
   END_RUNG
   RUNG wire#powerrail
      Contact( "Comm_ok" )
      { S7_Templates := "SrcType := Int" } EQ_Contact(in1 := "IEC_Counter_0_DB".CV, in2 := 20)
      I_Contact( "Modbus_Master_DB".BUSY )
   END_RUNG wire#w1
   // the same network as SCL:
   IF "IEC_Counter_0_DB".CV = 20 THEN
       "Modbus_Master_DB"(REQ := "Comm_ok" AND ("IEC_Counter_0_DB".CV = 20) AND NOT "Modbus_Master_DB".BUSY,   // Modbus_Master
                          MB_ADDR := 1,
                          MODE := 0,
                          DATA_ADDR := 32023,
                          DATA_LEN := 1,
                          DATA_PTR := "Modbus_Send_Receive_1".Reading_Struct."32023",
                          DONE => "Modbus".Done,
                          BUSY => "Modbus".Busy,
                          ERROR => "Modbus".Error,
                          STATUS => "Modbus".Status);
   END_IF;
END_REGION

REGION Network 26: RD 32025
   RUNG wire#powerrail
      { S7_Templates := "SrcType := Int" } EQ_Contact(in1 := "IEC_Counter_0_DB".CV, in2 := 21)
      { S7_Templates := "[card := 0, word_type := UInt, dword_type := UDInt, byte_type := USInt, any_type := Variant]" } "Modbus_Master_DB".Modbus_Master(REQ := wire#w1, MB_ADDR := 1, MODE := 0, DATA_ADDR := 32025, DATA_LEN := 1, DATA_PTR := "Modbus_Send_Receive_1".Reading_Struct."32025", DONE => "Modbus".Done, BUSY => "Modbus".Busy, ERROR => "Modbus".Error, STATUS => "Modbus".Status)
   END_RUNG
   RUNG wire#powerrail
      Contact( "Comm_ok" )
      { S7_Templates := "SrcType := Int" } EQ_Contact(in1 := "IEC_Counter_0_DB".CV, in2 := 21)
      I_Contact( "Modbus_Master_DB".BUSY )
   END_RUNG wire#w1
   // the same network as SCL:
   IF "IEC_Counter_0_DB".CV = 21 THEN
       "Modbus_Master_DB"(REQ := "Comm_ok" AND ("IEC_Counter_0_DB".CV = 21) AND NOT "Modbus_Master_DB".BUSY,   // Modbus_Master
                          MB_ADDR := 1,
                          MODE := 0,
                          DATA_ADDR := 32025,
                          DATA_LEN := 1,
                          DATA_PTR := "Modbus_Send_Receive_1".Reading_Struct."32025",
                          DONE => "Modbus".Done,
                          BUSY => "Modbus".Busy,
                          ERROR => "Modbus".Error,
                          STATUS => "Modbus".Status);
   END_IF;
END_REGION

REGION Network 27: RD 32026
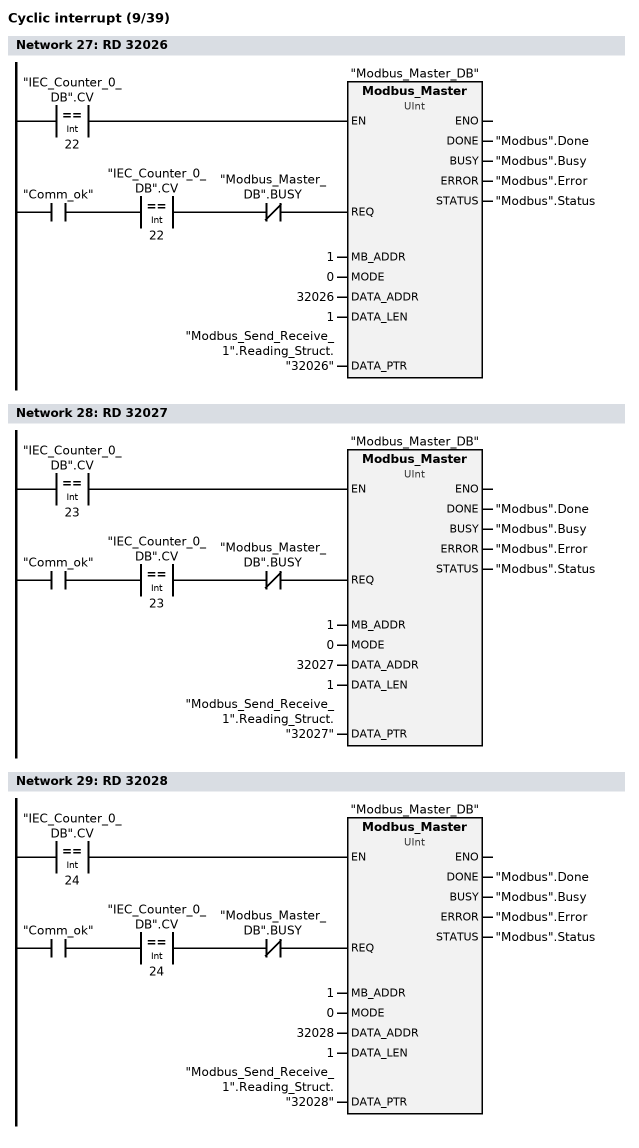
   RUNG wire#powerrail
      { S7_Templates := "SrcType := Int" } EQ_Contact(in1 := "IEC_Counter_0_DB".CV, in2 := 22)
      { S7_Templates := "[card := 0, word_type := UInt, dword_type := UDInt, byte_type := USInt, any_type := Variant]" } "Modbus_Master_DB".Modbus_Master(REQ := wire#w1, MB_ADDR := 1, MODE := 0, DATA_ADDR := 32026, DATA_LEN := 1, DATA_PTR := "Modbus_Send_Receive_1".Reading_Struct."32026", DONE => "Modbus".Done, BUSY => "Modbus".Busy, ERROR => "Modbus".Error, STATUS => "Modbus".Status)
   END_RUNG
   RUNG wire#powerrail
      Contact( "Comm_ok" )
      { S7_Templates := "SrcType := Int" } EQ_Contact(in1 := "IEC_Counter_0_DB".CV, in2 := 22)
      I_Contact( "Modbus_Master_DB".BUSY )
   END_RUNG wire#w1
   // the same network as SCL:
   IF "IEC_Counter_0_DB".CV = 22 THEN
       "Modbus_Master_DB"(REQ := "Comm_ok" AND ("IEC_Counter_0_DB".CV = 22) AND NOT "Modbus_Master_DB".BUSY,   // Modbus_Master
                          MB_ADDR := 1,
                          MODE := 0,
                          DATA_ADDR := 32026,
                          DATA_LEN := 1,
                          DATA_PTR := "Modbus_Send_Receive_1".Reading_Struct."32026",
                          DONE => "Modbus".Done,
                          BUSY => "Modbus".Busy,
                          ERROR => "Modbus".Error,
                          STATUS => "Modbus".Status);
   END_IF;
END_REGION

REGION Network 28: RD 32027
   RUNG wire#powerrail
      { S7_Templates := "SrcType := Int" } EQ_Contact(in1 := "IEC_Counter_0_DB".CV, in2 := 23)
      { S7_Templates := "[card := 0, word_type := UInt, dword_type := UDInt, byte_type := USInt, any_type := Variant]" } "Modbus_Master_DB".Modbus_Master(REQ := wire#w1, MB_ADDR := 1, MODE := 0, DATA_ADDR := 32027, DATA_LEN := 1, DATA_PTR := "Modbus_Send_Receive_1".Reading_Struct."32027", DONE => "Modbus".Done, BUSY => "Modbus".Busy, ERROR => "Modbus".Error, STATUS => "Modbus".Status)
   END_RUNG
   RUNG wire#powerrail
      Contact( "Comm_ok" )
      { S7_Templates := "SrcType := Int" } EQ_Contact(in1 := "IEC_Counter_0_DB".CV, in2 := 23)
      I_Contact( "Modbus_Master_DB".BUSY )
   END_RUNG wire#w1
   // the same network as SCL:
   IF "IEC_Counter_0_DB".CV = 23 THEN
       "Modbus_Master_DB"(REQ := "Comm_ok" AND ("IEC_Counter_0_DB".CV = 23) AND NOT "Modbus_Master_DB".BUSY,   // Modbus_Master
                          MB_ADDR := 1,
                          MODE := 0,
                          DATA_ADDR := 32027,
                          DATA_LEN := 1,
                          DATA_PTR := "Modbus_Send_Receive_1".Reading_Struct."32027",
                          DONE => "Modbus".Done,
                          BUSY => "Modbus".Busy,
                          ERROR => "Modbus".Error,
                          STATUS => "Modbus".Status);
   END_IF;
END_REGION

REGION Network 29: RD 32028
   RUNG wire#powerrail
      { S7_Templates := "SrcType := Int" } EQ_Contact(in1 := "IEC_Counter_0_DB".CV, in2 := 24)
      { S7_Templates := "[card := 0, word_type := UInt, dword_type := UDInt, byte_type := USInt, any_type := Variant]" } "Modbus_Master_DB".Modbus_Master(REQ := wire#w1, MB_ADDR := 1, MODE := 0, DATA_ADDR := 32028, DATA_LEN := 1, DATA_PTR := "Modbus_Send_Receive_1".Reading_Struct."32028", DONE => "Modbus".Done, BUSY => "Modbus".Busy, ERROR => "Modbus".Error, STATUS => "Modbus".Status)
   END_RUNG
   RUNG wire#powerrail
      Contact( "Comm_ok" )
      { S7_Templates := "SrcType := Int" } EQ_Contact(in1 := "IEC_Counter_0_DB".CV, in2 := 24)
      I_Contact( "Modbus_Master_DB".BUSY )
   END_RUNG wire#w1
   // the same network as SCL:
   IF "IEC_Counter_0_DB".CV = 24 THEN
       "Modbus_Master_DB"(REQ := "Comm_ok" AND ("IEC_Counter_0_DB".CV = 24) AND NOT "Modbus_Master_DB".BUSY,   // Modbus_Master
                          MB_ADDR := 1,
                          MODE := 0,
                          DATA_ADDR := 32028,
                          DATA_LEN := 1,
                          DATA_PTR := "Modbus_Send_Receive_1".Reading_Struct."32028",
                          DONE => "Modbus".Done,
                          BUSY => "Modbus".Busy,
                          ERROR => "Modbus".Error,
                          STATUS => "Modbus".Status);
   END_IF;
END_REGION

REGION Network 30: RD 32029
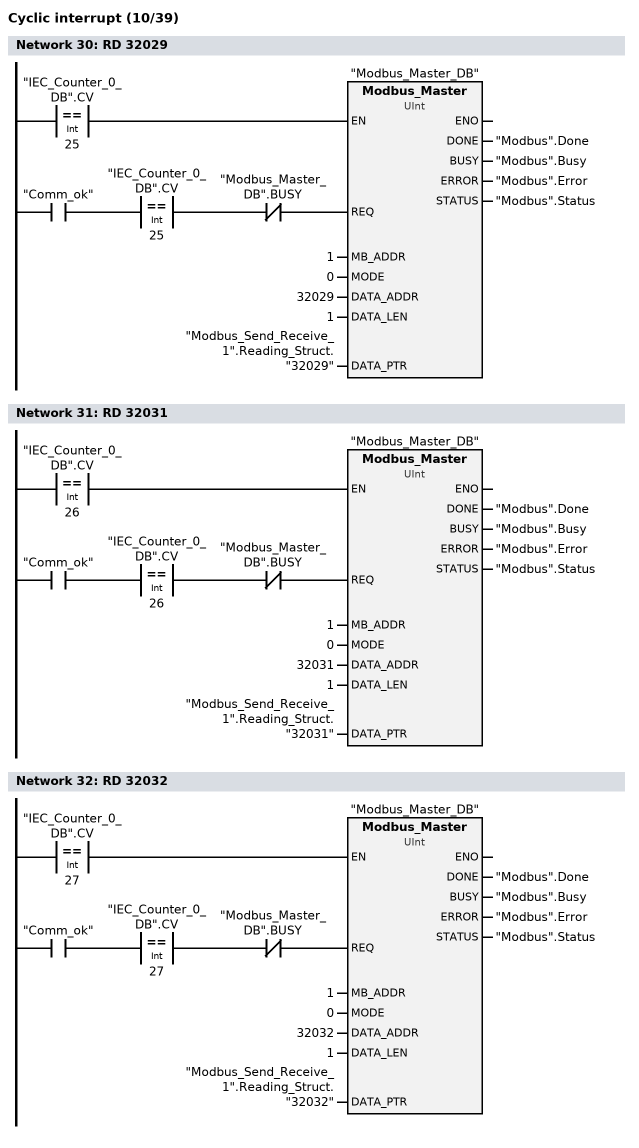
   RUNG wire#powerrail
      { S7_Templates := "SrcType := Int" } EQ_Contact(in1 := "IEC_Counter_0_DB".CV, in2 := 25)
      { S7_Templates := "[card := 0, word_type := UInt, dword_type := UDInt, byte_type := USInt, any_type := Variant]" } "Modbus_Master_DB".Modbus_Master(REQ := wire#w1, MB_ADDR := 1, MODE := 0, DATA_ADDR := 32029, DATA_LEN := 1, DATA_PTR := "Modbus_Send_Receive_1".Reading_Struct."32029", DONE => "Modbus".Done, BUSY => "Modbus".Busy, ERROR => "Modbus".Error, STATUS => "Modbus".Status)
   END_RUNG
   RUNG wire#powerrail
      Contact( "Comm_ok" )
      { S7_Templates := "SrcType := Int" } EQ_Contact(in1 := "IEC_Counter_0_DB".CV, in2 := 25)
      I_Contact( "Modbus_Master_DB".BUSY )
   END_RUNG wire#w1
   // the same network as SCL:
   IF "IEC_Counter_0_DB".CV = 25 THEN
       "Modbus_Master_DB"(REQ := "Comm_ok" AND ("IEC_Counter_0_DB".CV = 25) AND NOT "Modbus_Master_DB".BUSY,   // Modbus_Master
                          MB_ADDR := 1,
                          MODE := 0,
                          DATA_ADDR := 32029,
                          DATA_LEN := 1,
                          DATA_PTR := "Modbus_Send_Receive_1".Reading_Struct."32029",
                          DONE => "Modbus".Done,
                          BUSY => "Modbus".Busy,
                          ERROR => "Modbus".Error,
                          STATUS => "Modbus".Status);
   END_IF;
END_REGION

REGION Network 31: RD 32031
   RUNG wire#powerrail
      { S7_Templates := "SrcType := Int" } EQ_Contact(in1 := "IEC_Counter_0_DB".CV, in2 := 26)
      { S7_Templates := "[card := 0, word_type := UInt, dword_type := UDInt, byte_type := USInt, any_type := Variant]" } "Modbus_Master_DB".Modbus_Master(REQ := wire#w1, MB_ADDR := 1, MODE := 0, DATA_ADDR := 32031, DATA_LEN := 1, DATA_PTR := "Modbus_Send_Receive_1".Reading_Struct."32031", DONE => "Modbus".Done, BUSY => "Modbus".Busy, ERROR => "Modbus".Error, STATUS => "Modbus".Status)
   END_RUNG
   RUNG wire#powerrail
      Contact( "Comm_ok" )
      { S7_Templates := "SrcType := Int" } EQ_Contact(in1 := "IEC_Counter_0_DB".CV, in2 := 26)
      I_Contact( "Modbus_Master_DB".BUSY )
   END_RUNG wire#w1
   // the same network as SCL:
   IF "IEC_Counter_0_DB".CV = 26 THEN
       "Modbus_Master_DB"(REQ := "Comm_ok" AND ("IEC_Counter_0_DB".CV = 26) AND NOT "Modbus_Master_DB".BUSY,   // Modbus_Master
                          MB_ADDR := 1,
                          MODE := 0,
                          DATA_ADDR := 32031,
                          DATA_LEN := 1,
                          DATA_PTR := "Modbus_Send_Receive_1".Reading_Struct."32031",
                          DONE => "Modbus".Done,
                          BUSY => "Modbus".Busy,
                          ERROR => "Modbus".Error,
                          STATUS => "Modbus".Status);
   END_IF;
END_REGION

REGION Network 32: RD 32032
   RUNG wire#powerrail
      { S7_Templates := "SrcType := Int" } EQ_Contact(in1 := "IEC_Counter_0_DB".CV, in2 := 27)
      { S7_Templates := "[card := 0, word_type := UInt, dword_type := UDInt, byte_type := USInt, any_type := Variant]" } "Modbus_Master_DB".Modbus_Master(REQ := wire#w1, MB_ADDR := 1, MODE := 0, DATA_ADDR := 32032, DATA_LEN := 1, DATA_PTR := "Modbus_Send_Receive_1".Reading_Struct."32032", DONE => "Modbus".Done, BUSY => "Modbus".Busy, ERROR => "Modbus".Error, STATUS => "Modbus".Status)
   END_RUNG
   RUNG wire#powerrail
      Contact( "Comm_ok" )
      { S7_Templates := "SrcType := Int" } EQ_Contact(in1 := "IEC_Counter_0_DB".CV, in2 := 27)
      I_Contact( "Modbus_Master_DB".BUSY )
   END_RUNG wire#w1
   // the same network as SCL:
   IF "IEC_Counter_0_DB".CV = 27 THEN
       "Modbus_Master_DB"(REQ := "Comm_ok" AND ("IEC_Counter_0_DB".CV = 27) AND NOT "Modbus_Master_DB".BUSY,   // Modbus_Master
                          MB_ADDR := 1,
                          MODE := 0,
                          DATA_ADDR := 32032,
                          DATA_LEN := 1,
                          DATA_PTR := "Modbus_Send_Receive_1".Reading_Struct."32032",
                          DONE => "Modbus".Done,
                          BUSY => "Modbus".Busy,
                          ERROR => "Modbus".Error,
                          STATUS => "Modbus".Status);
   END_IF;
END_REGION

REGION Network 33: RD 32033
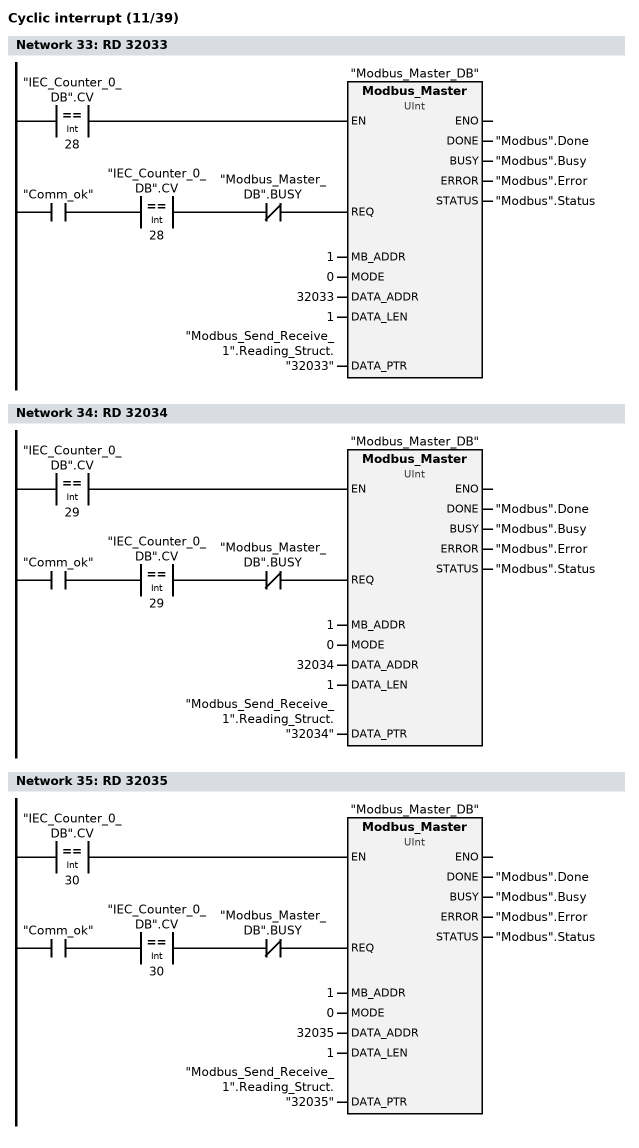
   RUNG wire#powerrail
      { S7_Templates := "SrcType := Int" } EQ_Contact(in1 := "IEC_Counter_0_DB".CV, in2 := 28)
      { S7_Templates := "[card := 0, word_type := UInt, dword_type := UDInt, byte_type := USInt, any_type := Variant]" } "Modbus_Master_DB".Modbus_Master(REQ := wire#w1, MB_ADDR := 1, MODE := 0, DATA_ADDR := 32033, DATA_LEN := 1, DATA_PTR := "Modbus_Send_Receive_1".Reading_Struct."32033", DONE => "Modbus".Done, BUSY => "Modbus".Busy, ERROR => "Modbus".Error, STATUS => "Modbus".Status)
   END_RUNG
   RUNG wire#powerrail
      Contact( "Comm_ok" )
      { S7_Templates := "SrcType := Int" } EQ_Contact(in1 := "IEC_Counter_0_DB".CV, in2 := 28)
      I_Contact( "Modbus_Master_DB".BUSY )
   END_RUNG wire#w1
   // the same network as SCL:
   IF "IEC_Counter_0_DB".CV = 28 THEN
       "Modbus_Master_DB"(REQ := "Comm_ok" AND ("IEC_Counter_0_DB".CV = 28) AND NOT "Modbus_Master_DB".BUSY,   // Modbus_Master
                          MB_ADDR := 1,
                          MODE := 0,
                          DATA_ADDR := 32033,
                          DATA_LEN := 1,
                          DATA_PTR := "Modbus_Send_Receive_1".Reading_Struct."32033",
                          DONE => "Modbus".Done,
                          BUSY => "Modbus".Busy,
                          ERROR => "Modbus".Error,
                          STATUS => "Modbus".Status);
   END_IF;
END_REGION

REGION Network 34: RD 32034
   RUNG wire#powerrail
      { S7_Templates := "SrcType := Int" } EQ_Contact(in1 := "IEC_Counter_0_DB".CV, in2 := 29)
      { S7_Templates := "[card := 0, word_type := UInt, dword_type := UDInt, byte_type := USInt, any_type := Variant]" } "Modbus_Master_DB".Modbus_Master(REQ := wire#w1, MB_ADDR := 1, MODE := 0, DATA_ADDR := 32034, DATA_LEN := 1, DATA_PTR := "Modbus_Send_Receive_1".Reading_Struct."32034", DONE => "Modbus".Done, BUSY => "Modbus".Busy, ERROR => "Modbus".Error, STATUS => "Modbus".Status)
   END_RUNG
   RUNG wire#powerrail
      Contact( "Comm_ok" )
      { S7_Templates := "SrcType := Int" } EQ_Contact(in1 := "IEC_Counter_0_DB".CV, in2 := 29)
      I_Contact( "Modbus_Master_DB".BUSY )
   END_RUNG wire#w1
   // the same network as SCL:
   IF "IEC_Counter_0_DB".CV = 29 THEN
       "Modbus_Master_DB"(REQ := "Comm_ok" AND ("IEC_Counter_0_DB".CV = 29) AND NOT "Modbus_Master_DB".BUSY,   // Modbus_Master
                          MB_ADDR := 1,
                          MODE := 0,
                          DATA_ADDR := 32034,
                          DATA_LEN := 1,
                          DATA_PTR := "Modbus_Send_Receive_1".Reading_Struct."32034",
                          DONE => "Modbus".Done,
                          BUSY => "Modbus".Busy,
                          ERROR => "Modbus".Error,
                          STATUS => "Modbus".Status);
   END_IF;
END_REGION

REGION Network 35: RD 32035
   RUNG wire#powerrail
      { S7_Templates := "SrcType := Int" } EQ_Contact(in1 := "IEC_Counter_0_DB".CV, in2 := 30)
      { S7_Templates := "[card := 0, word_type := UInt, dword_type := UDInt, byte_type := USInt, any_type := Variant]" } "Modbus_Master_DB".Modbus_Master(REQ := wire#w1, MB_ADDR := 1, MODE := 0, DATA_ADDR := 32035, DATA_LEN := 1, DATA_PTR := "Modbus_Send_Receive_1".Reading_Struct."32035", DONE => "Modbus".Done, BUSY => "Modbus".Busy, ERROR => "Modbus".Error, STATUS => "Modbus".Status)
   END_RUNG
   RUNG wire#powerrail
      Contact( "Comm_ok" )
      { S7_Templates := "SrcType := Int" } EQ_Contact(in1 := "IEC_Counter_0_DB".CV, in2 := 30)
      I_Contact( "Modbus_Master_DB".BUSY )
   END_RUNG wire#w1
   // the same network as SCL:
   IF "IEC_Counter_0_DB".CV = 30 THEN
       "Modbus_Master_DB"(REQ := "Comm_ok" AND ("IEC_Counter_0_DB".CV = 30) AND NOT "Modbus_Master_DB".BUSY,   // Modbus_Master
                          MB_ADDR := 1,
                          MODE := 0,
                          DATA_ADDR := 32035,
                          DATA_LEN := 1,
                          DATA_PTR := "Modbus_Send_Receive_1".Reading_Struct."32035",
                          DONE => "Modbus".Done,
                          BUSY => "Modbus".Busy,
                          ERROR => "Modbus".Error,
                          STATUS => "Modbus".Status);
   END_IF;
END_REGION

REGION Network 36: RD 32037
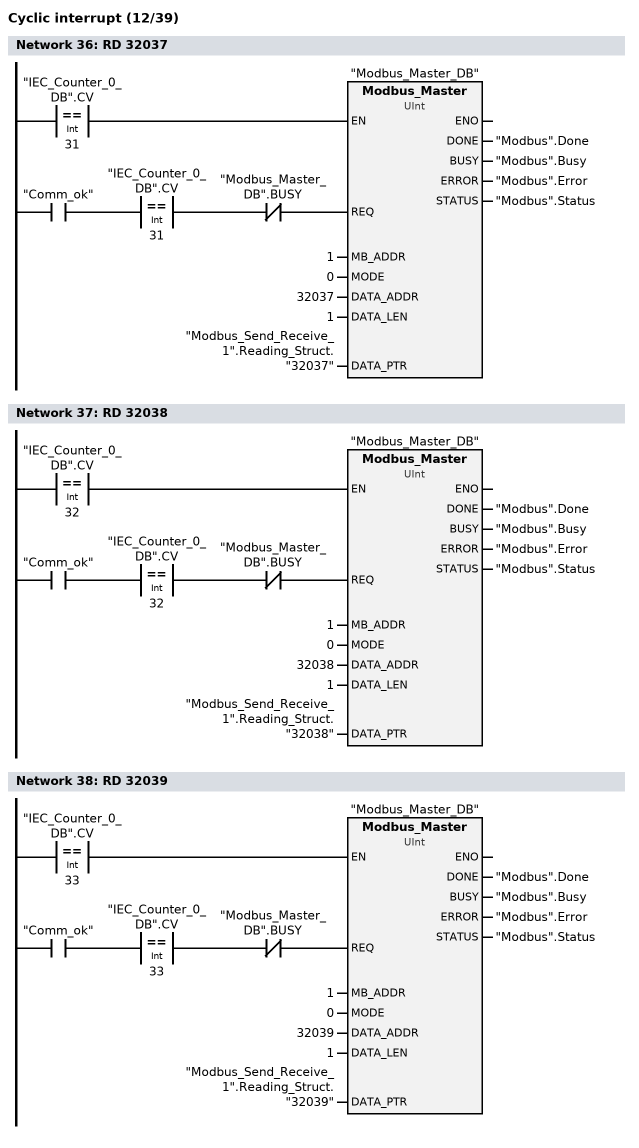
   RUNG wire#powerrail
      { S7_Templates := "SrcType := Int" } EQ_Contact(in1 := "IEC_Counter_0_DB".CV, in2 := 31)
      { S7_Templates := "[card := 0, word_type := UInt, dword_type := UDInt, byte_type := USInt, any_type := Variant]" } "Modbus_Master_DB".Modbus_Master(REQ := wire#w1, MB_ADDR := 1, MODE := 0, DATA_ADDR := 32037, DATA_LEN := 1, DATA_PTR := "Modbus_Send_Receive_1".Reading_Struct."32037", DONE => "Modbus".Done, BUSY => "Modbus".Busy, ERROR => "Modbus".Error, STATUS => "Modbus".Status)
   END_RUNG
   RUNG wire#powerrail
      Contact( "Comm_ok" )
      { S7_Templates := "SrcType := Int" } EQ_Contact(in1 := "IEC_Counter_0_DB".CV, in2 := 31)
      I_Contact( "Modbus_Master_DB".BUSY )
   END_RUNG wire#w1
   // the same network as SCL:
   IF "IEC_Counter_0_DB".CV = 31 THEN
       "Modbus_Master_DB"(REQ := "Comm_ok" AND ("IEC_Counter_0_DB".CV = 31) AND NOT "Modbus_Master_DB".BUSY,   // Modbus_Master
                          MB_ADDR := 1,
                          MODE := 0,
                          DATA_ADDR := 32037,
                          DATA_LEN := 1,
                          DATA_PTR := "Modbus_Send_Receive_1".Reading_Struct."32037",
                          DONE => "Modbus".Done,
                          BUSY => "Modbus".Busy,
                          ERROR => "Modbus".Error,
                          STATUS => "Modbus".Status);
   END_IF;
END_REGION

REGION Network 37: RD 32038
   RUNG wire#powerrail
      { S7_Templates := "SrcType := Int" } EQ_Contact(in1 := "IEC_Counter_0_DB".CV, in2 := 32)
      { S7_Templates := "[card := 0, word_type := UInt, dword_type := UDInt, byte_type := USInt, any_type := Variant]" } "Modbus_Master_DB".Modbus_Master(REQ := wire#w1, MB_ADDR := 1, MODE := 0, DATA_ADDR := 32038, DATA_LEN := 1, DATA_PTR := "Modbus_Send_Receive_1".Reading_Struct."32038", DONE => "Modbus".Done, BUSY => "Modbus".Busy, ERROR => "Modbus".Error, STATUS => "Modbus".Status)
   END_RUNG
   RUNG wire#powerrail
      Contact( "Comm_ok" )
      { S7_Templates := "SrcType := Int" } EQ_Contact(in1 := "IEC_Counter_0_DB".CV, in2 := 32)
      I_Contact( "Modbus_Master_DB".BUSY )
   END_RUNG wire#w1
   // the same network as SCL:
   IF "IEC_Counter_0_DB".CV = 32 THEN
       "Modbus_Master_DB"(REQ := "Comm_ok" AND ("IEC_Counter_0_DB".CV = 32) AND NOT "Modbus_Master_DB".BUSY,   // Modbus_Master
                          MB_ADDR := 1,
                          MODE := 0,
                          DATA_ADDR := 32038,
                          DATA_LEN := 1,
                          DATA_PTR := "Modbus_Send_Receive_1".Reading_Struct."32038",
                          DONE => "Modbus".Done,
                          BUSY => "Modbus".Busy,
                          ERROR => "Modbus".Error,
                          STATUS => "Modbus".Status);
   END_IF;
END_REGION

REGION Network 38: RD 32039
   RUNG wire#powerrail
      { S7_Templates := "SrcType := Int" } EQ_Contact(in1 := "IEC_Counter_0_DB".CV, in2 := 33)
      { S7_Templates := "[card := 0, word_type := UInt, dword_type := UDInt, byte_type := USInt, any_type := Variant]" } "Modbus_Master_DB".Modbus_Master(REQ := wire#w1, MB_ADDR := 1, MODE := 0, DATA_ADDR := 32039, DATA_LEN := 1, DATA_PTR := "Modbus_Send_Receive_1".Reading_Struct."32039", DONE => "Modbus".Done, BUSY => "Modbus".Busy, ERROR => "Modbus".Error, STATUS => "Modbus".Status)
   END_RUNG
   RUNG wire#powerrail
      Contact( "Comm_ok" )
      { S7_Templates := "SrcType := Int" } EQ_Contact(in1 := "IEC_Counter_0_DB".CV, in2 := 33)
      I_Contact( "Modbus_Master_DB".BUSY )
   END_RUNG wire#w1
   // the same network as SCL:
   IF "IEC_Counter_0_DB".CV = 33 THEN
       "Modbus_Master_DB"(REQ := "Comm_ok" AND ("IEC_Counter_0_DB".CV = 33) AND NOT "Modbus_Master_DB".BUSY,   // Modbus_Master
                          MB_ADDR := 1,
                          MODE := 0,
                          DATA_ADDR := 32039,
                          DATA_LEN := 1,
                          DATA_PTR := "Modbus_Send_Receive_1".Reading_Struct."32039",
                          DONE => "Modbus".Done,
                          BUSY => "Modbus".Busy,
                          ERROR => "Modbus".Error,
                          STATUS => "Modbus".Status);
   END_IF;
END_REGION

REGION Network 39: RD 32040
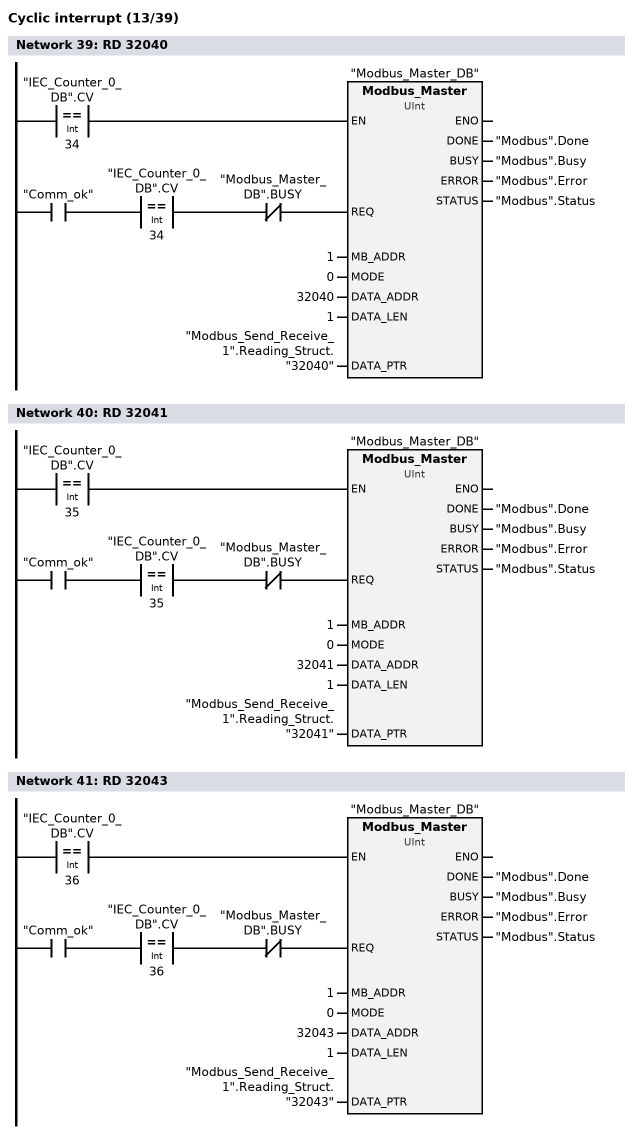
   RUNG wire#powerrail
      { S7_Templates := "SrcType := Int" } EQ_Contact(in1 := "IEC_Counter_0_DB".CV, in2 := 34)
      { S7_Templates := "[card := 0, word_type := UInt, dword_type := UDInt, byte_type := USInt, any_type := Variant]" } "Modbus_Master_DB".Modbus_Master(REQ := wire#w1, MB_ADDR := 1, MODE := 0, DATA_ADDR := 32040, DATA_LEN := 1, DATA_PTR := "Modbus_Send_Receive_1".Reading_Struct."32040", DONE => "Modbus".Done, BUSY => "Modbus".Busy, ERROR => "Modbus".Error, STATUS => "Modbus".Status)
   END_RUNG
   RUNG wire#powerrail
      Contact( "Comm_ok" )
      { S7_Templates := "SrcType := Int" } EQ_Contact(in1 := "IEC_Counter_0_DB".CV, in2 := 34)
      I_Contact( "Modbus_Master_DB".BUSY )
   END_RUNG wire#w1
   // the same network as SCL:
   IF "IEC_Counter_0_DB".CV = 34 THEN
       "Modbus_Master_DB"(REQ := "Comm_ok" AND ("IEC_Counter_0_DB".CV = 34) AND NOT "Modbus_Master_DB".BUSY,   // Modbus_Master
                          MB_ADDR := 1,
                          MODE := 0,
                          DATA_ADDR := 32040,
                          DATA_LEN := 1,
                          DATA_PTR := "Modbus_Send_Receive_1".Reading_Struct."32040",
                          DONE => "Modbus".Done,
                          BUSY => "Modbus".Busy,
                          ERROR => "Modbus".Error,
                          STATUS => "Modbus".Status);
   END_IF;
END_REGION

REGION Network 40: RD 32041
   RUNG wire#powerrail
      { S7_Templates := "SrcType := Int" } EQ_Contact(in1 := "IEC_Counter_0_DB".CV, in2 := 35)
      { S7_Templates := "[card := 0, word_type := UInt, dword_type := UDInt, byte_type := USInt, any_type := Variant]" } "Modbus_Master_DB".Modbus_Master(REQ := wire#w1, MB_ADDR := 1, MODE := 0, DATA_ADDR := 32041, DATA_LEN := 1, DATA_PTR := "Modbus_Send_Receive_1".Reading_Struct."32041", DONE => "Modbus".Done, BUSY => "Modbus".Busy, ERROR => "Modbus".Error, STATUS => "Modbus".Status)
   END_RUNG
   RUNG wire#powerrail
      Contact( "Comm_ok" )
      { S7_Templates := "SrcType := Int" } EQ_Contact(in1 := "IEC_Counter_0_DB".CV, in2 := 35)
      I_Contact( "Modbus_Master_DB".BUSY )
   END_RUNG wire#w1
   // the same network as SCL:
   IF "IEC_Counter_0_DB".CV = 35 THEN
       "Modbus_Master_DB"(REQ := "Comm_ok" AND ("IEC_Counter_0_DB".CV = 35) AND NOT "Modbus_Master_DB".BUSY,   // Modbus_Master
                          MB_ADDR := 1,
                          MODE := 0,
                          DATA_ADDR := 32041,
                          DATA_LEN := 1,
                          DATA_PTR := "Modbus_Send_Receive_1".Reading_Struct."32041",
                          DONE => "Modbus".Done,
                          BUSY => "Modbus".Busy,
                          ERROR => "Modbus".Error,
                          STATUS => "Modbus".Status);
   END_IF;
END_REGION

REGION Network 41: RD 32043
   RUNG wire#powerrail
      { S7_Templates := "SrcType := Int" } EQ_Contact(in1 := "IEC_Counter_0_DB".CV, in2 := 36)
      { S7_Templates := "[card := 0, word_type := UInt, dword_type := UDInt, byte_type := USInt, any_type := Variant]" } "Modbus_Master_DB".Modbus_Master(REQ := wire#w1, MB_ADDR := 1, MODE := 0, DATA_ADDR := 32043, DATA_LEN := 1, DATA_PTR := "Modbus_Send_Receive_1".Reading_Struct."32043", DONE => "Modbus".Done, BUSY => "Modbus".Busy, ERROR => "Modbus".Error, STATUS => "Modbus".Status)
   END_RUNG
   RUNG wire#powerrail
      Contact( "Comm_ok" )
      { S7_Templates := "SrcType := Int" } EQ_Contact(in1 := "IEC_Counter_0_DB".CV, in2 := 36)
      I_Contact( "Modbus_Master_DB".BUSY )
   END_RUNG wire#w1
   // the same network as SCL:
   IF "IEC_Counter_0_DB".CV = 36 THEN
       "Modbus_Master_DB"(REQ := "Comm_ok" AND ("IEC_Counter_0_DB".CV = 36) AND NOT "Modbus_Master_DB".BUSY,   // Modbus_Master
                          MB_ADDR := 1,
                          MODE := 0,
                          DATA_ADDR := 32043,
                          DATA_LEN := 1,
                          DATA_PTR := "Modbus_Send_Receive_1".Reading_Struct."32043",
                          DONE => "Modbus".Done,
                          BUSY => "Modbus".Busy,
                          ERROR => "Modbus".Error,
                          STATUS => "Modbus".Status);
   END_IF;
END_REGION

REGION Network 42: RD 32044
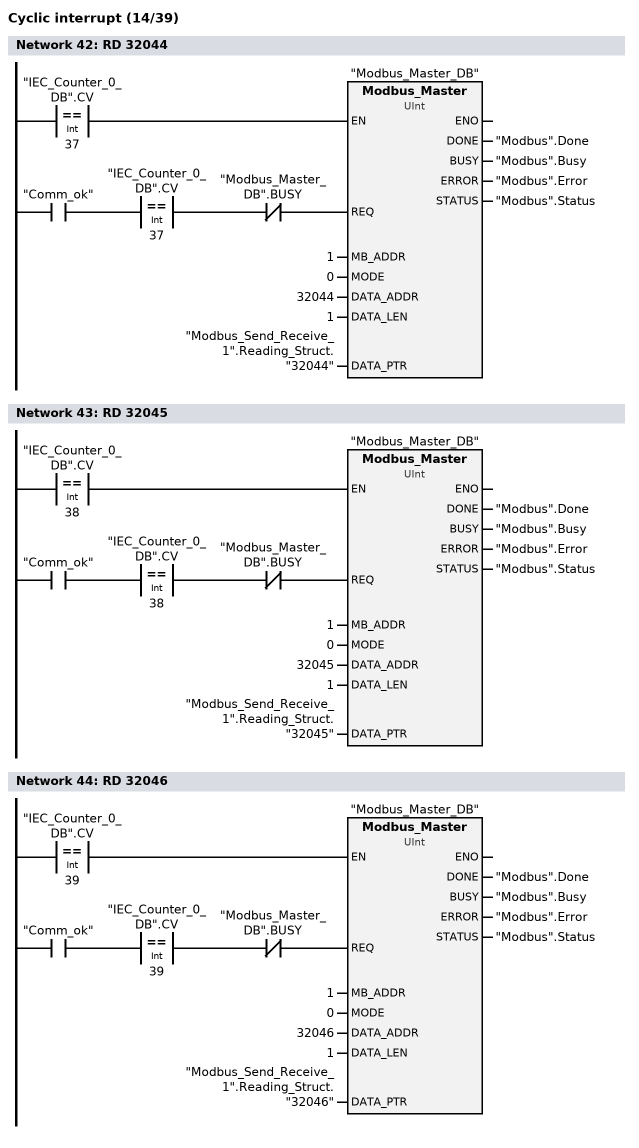
   RUNG wire#powerrail
      { S7_Templates := "SrcType := Int" } EQ_Contact(in1 := "IEC_Counter_0_DB".CV, in2 := 37)
      { S7_Templates := "[card := 0, word_type := UInt, dword_type := UDInt, byte_type := USInt, any_type := Variant]" } "Modbus_Master_DB".Modbus_Master(REQ := wire#w1, MB_ADDR := 1, MODE := 0, DATA_ADDR := 32044, DATA_LEN := 1, DATA_PTR := "Modbus_Send_Receive_1".Reading_Struct."32044", DONE => "Modbus".Done, BUSY => "Modbus".Busy, ERROR => "Modbus".Error, STATUS => "Modbus".Status)
   END_RUNG
   RUNG wire#powerrail
      Contact( "Comm_ok" )
      { S7_Templates := "SrcType := Int" } EQ_Contact(in1 := "IEC_Counter_0_DB".CV, in2 := 37)
      I_Contact( "Modbus_Master_DB".BUSY )
   END_RUNG wire#w1
   // the same network as SCL:
   IF "IEC_Counter_0_DB".CV = 37 THEN
       "Modbus_Master_DB"(REQ := "Comm_ok" AND ("IEC_Counter_0_DB".CV = 37) AND NOT "Modbus_Master_DB".BUSY,   // Modbus_Master
                          MB_ADDR := 1,
                          MODE := 0,
                          DATA_ADDR := 32044,
                          DATA_LEN := 1,
                          DATA_PTR := "Modbus_Send_Receive_1".Reading_Struct."32044",
                          DONE => "Modbus".Done,
                          BUSY => "Modbus".Busy,
                          ERROR => "Modbus".Error,
                          STATUS => "Modbus".Status);
   END_IF;
END_REGION

REGION Network 43: RD 32045
   RUNG wire#powerrail
      { S7_Templates := "SrcType := Int" } EQ_Contact(in1 := "IEC_Counter_0_DB".CV, in2 := 38)
      { S7_Templates := "[card := 0, word_type := UInt, dword_type := UDInt, byte_type := USInt, any_type := Variant]" } "Modbus_Master_DB".Modbus_Master(REQ := wire#w1, MB_ADDR := 1, MODE := 0, DATA_ADDR := 32045, DATA_LEN := 1, DATA_PTR := "Modbus_Send_Receive_1".Reading_Struct."32045", DONE => "Modbus".Done, BUSY => "Modbus".Busy, ERROR => "Modbus".Error, STATUS => "Modbus".Status)
   END_RUNG
   RUNG wire#powerrail
      Contact( "Comm_ok" )
      { S7_Templates := "SrcType := Int" } EQ_Contact(in1 := "IEC_Counter_0_DB".CV, in2 := 38)
      I_Contact( "Modbus_Master_DB".BUSY )
   END_RUNG wire#w1
   // the same network as SCL:
   IF "IEC_Counter_0_DB".CV = 38 THEN
       "Modbus_Master_DB"(REQ := "Comm_ok" AND ("IEC_Counter_0_DB".CV = 38) AND NOT "Modbus_Master_DB".BUSY,   // Modbus_Master
                          MB_ADDR := 1,
                          MODE := 0,
                          DATA_ADDR := 32045,
                          DATA_LEN := 1,
                          DATA_PTR := "Modbus_Send_Receive_1".Reading_Struct."32045",
                          DONE => "Modbus".Done,
                          BUSY => "Modbus".Busy,
                          ERROR => "Modbus".Error,
                          STATUS => "Modbus".Status);
   END_IF;
END_REGION

REGION Network 44: RD 32046
   RUNG wire#powerrail
      { S7_Templates := "SrcType := Int" } EQ_Contact(in1 := "IEC_Counter_0_DB".CV, in2 := 39)
      { S7_Templates := "[card := 0, word_type := UInt, dword_type := UDInt, byte_type := USInt, any_type := Variant]" } "Modbus_Master_DB".Modbus_Master(REQ := wire#w1, MB_ADDR := 1, MODE := 0, DATA_ADDR := 32046, DATA_LEN := 1, DATA_PTR := "Modbus_Send_Receive_1".Reading_Struct."32046", DONE => "Modbus".Done, BUSY => "Modbus".Busy, ERROR => "Modbus".Error, STATUS => "Modbus".Status)
   END_RUNG
   RUNG wire#powerrail
      Contact( "Comm_ok" )
      { S7_Templates := "SrcType := Int" } EQ_Contact(in1 := "IEC_Counter_0_DB".CV, in2 := 39)
      I_Contact( "Modbus_Master_DB".BUSY )
   END_RUNG wire#w1
   // the same network as SCL:
   IF "IEC_Counter_0_DB".CV = 39 THEN
       "Modbus_Master_DB"(REQ := "Comm_ok" AND ("IEC_Counter_0_DB".CV = 39) AND NOT "Modbus_Master_DB".BUSY,   // Modbus_Master
                          MB_ADDR := 1,
                          MODE := 0,
                          DATA_ADDR := 32046,
                          DATA_LEN := 1,
                          DATA_PTR := "Modbus_Send_Receive_1".Reading_Struct."32046",
                          DONE => "Modbus".Done,
                          BUSY => "Modbus".Busy,
                          ERROR => "Modbus".Error,
                          STATUS => "Modbus".Status);
   END_IF;
END_REGION

REGION Network 45: RD 32047
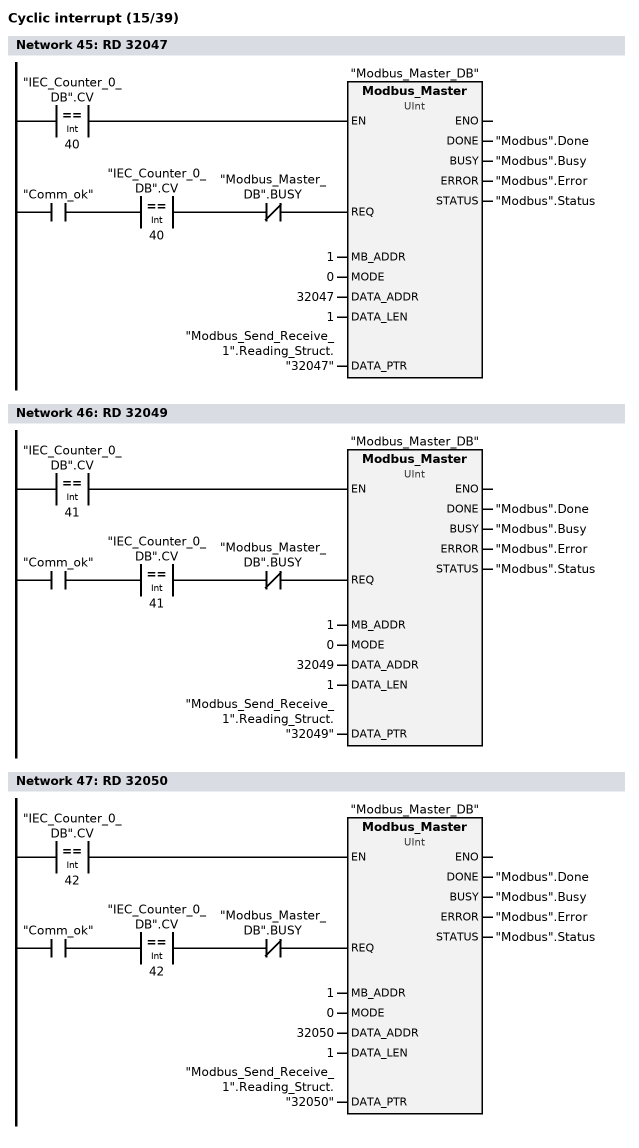
   RUNG wire#powerrail
      { S7_Templates := "SrcType := Int" } EQ_Contact(in1 := "IEC_Counter_0_DB".CV, in2 := 40)
      { S7_Templates := "[card := 0, word_type := UInt, dword_type := UDInt, byte_type := USInt, any_type := Variant]" } "Modbus_Master_DB".Modbus_Master(REQ := wire#w1, MB_ADDR := 1, MODE := 0, DATA_ADDR := 32047, DATA_LEN := 1, DATA_PTR := "Modbus_Send_Receive_1".Reading_Struct."32047", DONE => "Modbus".Done, BUSY => "Modbus".Busy, ERROR => "Modbus".Error, STATUS => "Modbus".Status)
   END_RUNG
   RUNG wire#powerrail
      Contact( "Comm_ok" )
      { S7_Templates := "SrcType := Int" } EQ_Contact(in1 := "IEC_Counter_0_DB".CV, in2 := 40)
      I_Contact( "Modbus_Master_DB".BUSY )
   END_RUNG wire#w1
   // the same network as SCL:
   IF "IEC_Counter_0_DB".CV = 40 THEN
       "Modbus_Master_DB"(REQ := "Comm_ok" AND ("IEC_Counter_0_DB".CV = 40) AND NOT "Modbus_Master_DB".BUSY,   // Modbus_Master
                          MB_ADDR := 1,
                          MODE := 0,
                          DATA_ADDR := 32047,
                          DATA_LEN := 1,
                          DATA_PTR := "Modbus_Send_Receive_1".Reading_Struct."32047",
                          DONE => "Modbus".Done,
                          BUSY => "Modbus".Busy,
                          ERROR => "Modbus".Error,
                          STATUS => "Modbus".Status);
   END_IF;
END_REGION

REGION Network 46: RD 32049
   RUNG wire#powerrail
      { S7_Templates := "SrcType := Int" } EQ_Contact(in1 := "IEC_Counter_0_DB".CV, in2 := 41)
      { S7_Templates := "[card := 0, word_type := UInt, dword_type := UDInt, byte_type := USInt, any_type := Variant]" } "Modbus_Master_DB".Modbus_Master(REQ := wire#w1, MB_ADDR := 1, MODE := 0, DATA_ADDR := 32049, DATA_LEN := 1, DATA_PTR := "Modbus_Send_Receive_1".Reading_Struct."32049", DONE => "Modbus".Done, BUSY => "Modbus".Busy, ERROR => "Modbus".Error, STATUS => "Modbus".Status)
   END_RUNG
   RUNG wire#powerrail
      Contact( "Comm_ok" )
      { S7_Templates := "SrcType := Int" } EQ_Contact(in1 := "IEC_Counter_0_DB".CV, in2 := 41)
      I_Contact( "Modbus_Master_DB".BUSY )
   END_RUNG wire#w1
   // the same network as SCL:
   IF "IEC_Counter_0_DB".CV = 41 THEN
       "Modbus_Master_DB"(REQ := "Comm_ok" AND ("IEC_Counter_0_DB".CV = 41) AND NOT "Modbus_Master_DB".BUSY,   // Modbus_Master
                          MB_ADDR := 1,
                          MODE := 0,
                          DATA_ADDR := 32049,
                          DATA_LEN := 1,
                          DATA_PTR := "Modbus_Send_Receive_1".Reading_Struct."32049",
                          DONE => "Modbus".Done,
                          BUSY => "Modbus".Busy,
                          ERROR => "Modbus".Error,
                          STATUS => "Modbus".Status);
   END_IF;
END_REGION

REGION Network 47: RD 32050
   RUNG wire#powerrail
      { S7_Templates := "SrcType := Int" } EQ_Contact(in1 := "IEC_Counter_0_DB".CV, in2 := 42)
      { S7_Templates := "[card := 0, word_type := UInt, dword_type := UDInt, byte_type := USInt, any_type := Variant]" } "Modbus_Master_DB".Modbus_Master(REQ := wire#w1, MB_ADDR := 1, MODE := 0, DATA_ADDR := 32050, DATA_LEN := 1, DATA_PTR := "Modbus_Send_Receive_1".Reading_Struct."32050", DONE => "Modbus".Done, BUSY => "Modbus".Busy, ERROR => "Modbus".Error, STATUS => "Modbus".Status)
   END_RUNG
   RUNG wire#powerrail
      Contact( "Comm_ok" )
      { S7_Templates := "SrcType := Int" } EQ_Contact(in1 := "IEC_Counter_0_DB".CV, in2 := 42)
      I_Contact( "Modbus_Master_DB".BUSY )
   END_RUNG wire#w1
   // the same network as SCL:
   IF "IEC_Counter_0_DB".CV = 42 THEN
       "Modbus_Master_DB"(REQ := "Comm_ok" AND ("IEC_Counter_0_DB".CV = 42) AND NOT "Modbus_Master_DB".BUSY,   // Modbus_Master
                          MB_ADDR := 1,
                          MODE := 0,
                          DATA_ADDR := 32050,
                          DATA_LEN := 1,
                          DATA_PTR := "Modbus_Send_Receive_1".Reading_Struct."32050",
                          DONE => "Modbus".Done,
                          BUSY => "Modbus".Busy,
                          ERROR => "Modbus".Error,
                          STATUS => "Modbus".Status);
   END_IF;
END_REGION

REGION Network 48: RD 32051
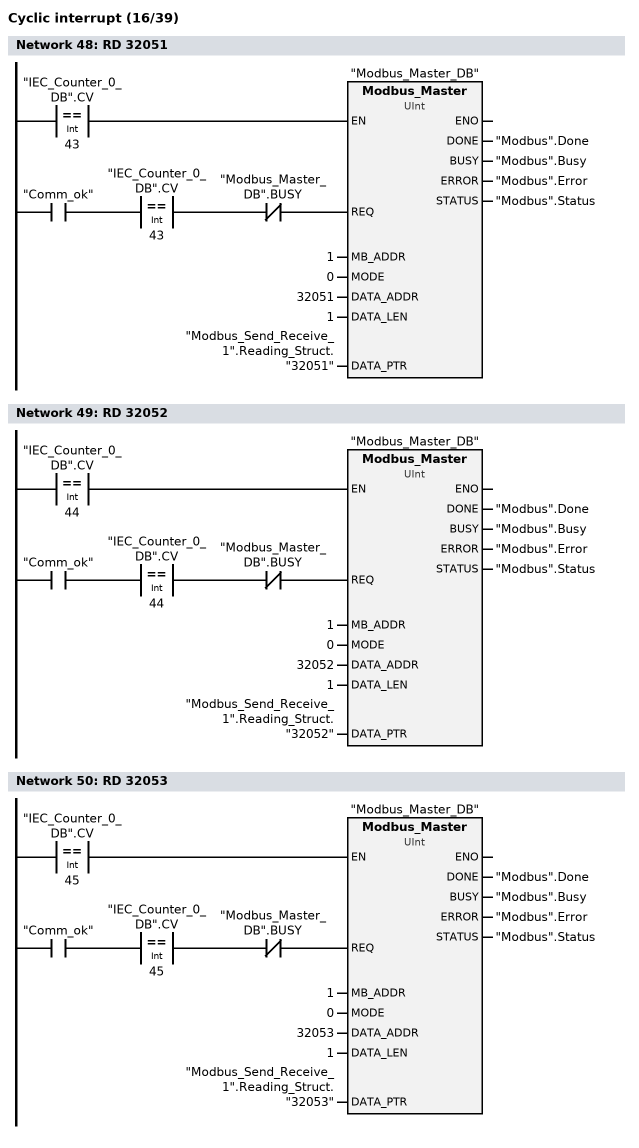
   RUNG wire#powerrail
      { S7_Templates := "SrcType := Int" } EQ_Contact(in1 := "IEC_Counter_0_DB".CV, in2 := 43)
      { S7_Templates := "[card := 0, word_type := UInt, dword_type := UDInt, byte_type := USInt, any_type := Variant]" } "Modbus_Master_DB".Modbus_Master(REQ := wire#w1, MB_ADDR := 1, MODE := 0, DATA_ADDR := 32051, DATA_LEN := 1, DATA_PTR := "Modbus_Send_Receive_1".Reading_Struct."32051", DONE => "Modbus".Done, BUSY => "Modbus".Busy, ERROR => "Modbus".Error, STATUS => "Modbus".Status)
   END_RUNG
   RUNG wire#powerrail
      Contact( "Comm_ok" )
      { S7_Templates := "SrcType := Int" } EQ_Contact(in1 := "IEC_Counter_0_DB".CV, in2 := 43)
      I_Contact( "Modbus_Master_DB".BUSY )
   END_RUNG wire#w1
   // the same network as SCL:
   IF "IEC_Counter_0_DB".CV = 43 THEN
       "Modbus_Master_DB"(REQ := "Comm_ok" AND ("IEC_Counter_0_DB".CV = 43) AND NOT "Modbus_Master_DB".BUSY,   // Modbus_Master
                          MB_ADDR := 1,
                          MODE := 0,
                          DATA_ADDR := 32051,
                          DATA_LEN := 1,
                          DATA_PTR := "Modbus_Send_Receive_1".Reading_Struct."32051",
                          DONE => "Modbus".Done,
                          BUSY => "Modbus".Busy,
                          ERROR => "Modbus".Error,
                          STATUS => "Modbus".Status);
   END_IF;
END_REGION

REGION Network 49: RD 32052
   RUNG wire#powerrail
      { S7_Templates := "SrcType := Int" } EQ_Contact(in1 := "IEC_Counter_0_DB".CV, in2 := 44)
      { S7_Templates := "[card := 0, word_type := UInt, dword_type := UDInt, byte_type := USInt, any_type := Variant]" } "Modbus_Master_DB".Modbus_Master(REQ := wire#w1, MB_ADDR := 1, MODE := 0, DATA_ADDR := 32052, DATA_LEN := 1, DATA_PTR := "Modbus_Send_Receive_1".Reading_Struct."32052", DONE => "Modbus".Done, BUSY => "Modbus".Busy, ERROR => "Modbus".Error, STATUS => "Modbus".Status)
   END_RUNG
   RUNG wire#powerrail
      Contact( "Comm_ok" )
      { S7_Templates := "SrcType := Int" } EQ_Contact(in1 := "IEC_Counter_0_DB".CV, in2 := 44)
      I_Contact( "Modbus_Master_DB".BUSY )
   END_RUNG wire#w1
   // the same network as SCL:
   IF "IEC_Counter_0_DB".CV = 44 THEN
       "Modbus_Master_DB"(REQ := "Comm_ok" AND ("IEC_Counter_0_DB".CV = 44) AND NOT "Modbus_Master_DB".BUSY,   // Modbus_Master
                          MB_ADDR := 1,
                          MODE := 0,
                          DATA_ADDR := 32052,
                          DATA_LEN := 1,
                          DATA_PTR := "Modbus_Send_Receive_1".Reading_Struct."32052",
                          DONE => "Modbus".Done,
                          BUSY => "Modbus".Busy,
                          ERROR => "Modbus".Error,
                          STATUS => "Modbus".Status);
   END_IF;
END_REGION

REGION Network 50: RD 32053
   RUNG wire#powerrail
      { S7_Templates := "SrcType := Int" } EQ_Contact(in1 := "IEC_Counter_0_DB".CV, in2 := 45)
      { S7_Templates := "[card := 0, word_type := UInt, dword_type := UDInt, byte_type := USInt, any_type := Variant]" } "Modbus_Master_DB".Modbus_Master(REQ := wire#w1, MB_ADDR := 1, MODE := 0, DATA_ADDR := 32053, DATA_LEN := 1, DATA_PTR := "Modbus_Send_Receive_1".Reading_Struct."32053", DONE => "Modbus".Done, BUSY => "Modbus".Busy, ERROR => "Modbus".Error, STATUS => "Modbus".Status)
   END_RUNG
   RUNG wire#powerrail
      Contact( "Comm_ok" )
      { S7_Templates := "SrcType := Int" } EQ_Contact(in1 := "IEC_Counter_0_DB".CV, in2 := 45)
      I_Contact( "Modbus_Master_DB".BUSY )
   END_RUNG wire#w1
   // the same network as SCL:
   IF "IEC_Counter_0_DB".CV = 45 THEN
       "Modbus_Master_DB"(REQ := "Comm_ok" AND ("IEC_Counter_0_DB".CV = 45) AND NOT "Modbus_Master_DB".BUSY,   // Modbus_Master
                          MB_ADDR := 1,
                          MODE := 0,
                          DATA_ADDR := 32053,
                          DATA_LEN := 1,
                          DATA_PTR := "Modbus_Send_Receive_1".Reading_Struct."32053",
                          DONE => "Modbus".Done,
                          BUSY => "Modbus".Busy,
                          ERROR => "Modbus".Error,
                          STATUS => "Modbus".Status);
   END_IF;
END_REGION

REGION Network 51: RD 32055
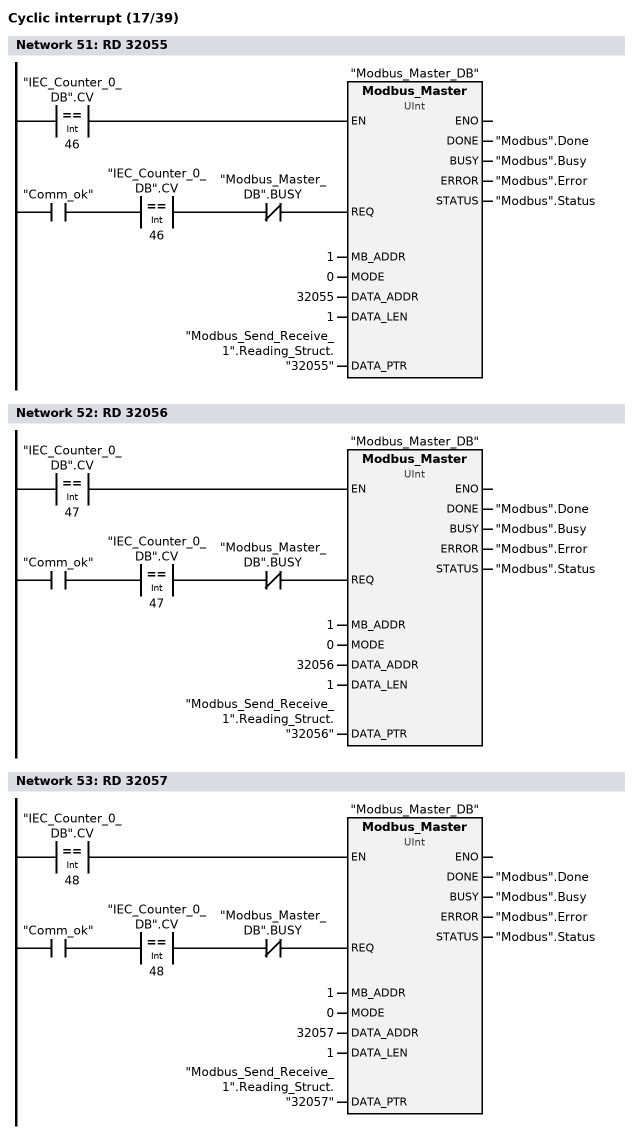
   RUNG wire#powerrail
      { S7_Templates := "SrcType := Int" } EQ_Contact(in1 := "IEC_Counter_0_DB".CV, in2 := 46)
      { S7_Templates := "[card := 0, word_type := UInt, dword_type := UDInt, byte_type := USInt, any_type := Variant]" } "Modbus_Master_DB".Modbus_Master(REQ := wire#w1, MB_ADDR := 1, MODE := 0, DATA_ADDR := 32055, DATA_LEN := 1, DATA_PTR := "Modbus_Send_Receive_1".Reading_Struct."32055", DONE => "Modbus".Done, BUSY => "Modbus".Busy, ERROR => "Modbus".Error, STATUS => "Modbus".Status)
   END_RUNG
   RUNG wire#powerrail
      Contact( "Comm_ok" )
      { S7_Templates := "SrcType := Int" } EQ_Contact(in1 := "IEC_Counter_0_DB".CV, in2 := 46)
      I_Contact( "Modbus_Master_DB".BUSY )
   END_RUNG wire#w1
   // the same network as SCL:
   IF "IEC_Counter_0_DB".CV = 46 THEN
       "Modbus_Master_DB"(REQ := "Comm_ok" AND ("IEC_Counter_0_DB".CV = 46) AND NOT "Modbus_Master_DB".BUSY,   // Modbus_Master
                          MB_ADDR := 1,
                          MODE := 0,
                          DATA_ADDR := 32055,
                          DATA_LEN := 1,
                          DATA_PTR := "Modbus_Send_Receive_1".Reading_Struct."32055",
                          DONE => "Modbus".Done,
                          BUSY => "Modbus".Busy,
                          ERROR => "Modbus".Error,
                          STATUS => "Modbus".Status);
   END_IF;
END_REGION

REGION Network 52: RD 32056
   RUNG wire#powerrail
      { S7_Templates := "SrcType := Int" } EQ_Contact(in1 := "IEC_Counter_0_DB".CV, in2 := 47)
      { S7_Templates := "[card := 0, word_type := UInt, dword_type := UDInt, byte_type := USInt, any_type := Variant]" } "Modbus_Master_DB".Modbus_Master(REQ := wire#w1, MB_ADDR := 1, MODE := 0, DATA_ADDR := 32056, DATA_LEN := 1, DATA_PTR := "Modbus_Send_Receive_1".Reading_Struct."32056", DONE => "Modbus".Done, BUSY => "Modbus".Busy, ERROR => "Modbus".Error, STATUS => "Modbus".Status)
   END_RUNG
   RUNG wire#powerrail
      Contact( "Comm_ok" )
      { S7_Templates := "SrcType := Int" } EQ_Contact(in1 := "IEC_Counter_0_DB".CV, in2 := 47)
      I_Contact( "Modbus_Master_DB".BUSY )
   END_RUNG wire#w1
   // the same network as SCL:
   IF "IEC_Counter_0_DB".CV = 47 THEN
       "Modbus_Master_DB"(REQ := "Comm_ok" AND ("IEC_Counter_0_DB".CV = 47) AND NOT "Modbus_Master_DB".BUSY,   // Modbus_Master
                          MB_ADDR := 1,
                          MODE := 0,
                          DATA_ADDR := 32056,
                          DATA_LEN := 1,
                          DATA_PTR := "Modbus_Send_Receive_1".Reading_Struct."32056",
                          DONE => "Modbus".Done,
                          BUSY => "Modbus".Busy,
                          ERROR => "Modbus".Error,
                          STATUS => "Modbus".Status);
   END_IF;
END_REGION

REGION Network 53: RD 32057
   RUNG wire#powerrail
      { S7_Templates := "SrcType := Int" } EQ_Contact(in1 := "IEC_Counter_0_DB".CV, in2 := 48)
      { S7_Templates := "[card := 0, word_type := UInt, dword_type := UDInt, byte_type := USInt, any_type := Variant]" } "Modbus_Master_DB".Modbus_Master(REQ := wire#w1, MB_ADDR := 1, MODE := 0, DATA_ADDR := 32057, DATA_LEN := 1, DATA_PTR := "Modbus_Send_Receive_1".Reading_Struct."32057", DONE => "Modbus".Done, BUSY => "Modbus".Busy, ERROR => "Modbus".Error, STATUS => "Modbus".Status)
   END_RUNG
   RUNG wire#powerrail
      Contact( "Comm_ok" )
      { S7_Templates := "SrcType := Int" } EQ_Contact(in1 := "IEC_Counter_0_DB".CV, in2 := 48)
      I_Contact( "Modbus_Master_DB".BUSY )
   END_RUNG wire#w1
   // the same network as SCL:
   IF "IEC_Counter_0_DB".CV = 48 THEN
       "Modbus_Master_DB"(REQ := "Comm_ok" AND ("IEC_Counter_0_DB".CV = 48) AND NOT "Modbus_Master_DB".BUSY,   // Modbus_Master
                          MB_ADDR := 1,
                          MODE := 0,
                          DATA_ADDR := 32057,
                          DATA_LEN := 1,
                          DATA_PTR := "Modbus_Send_Receive_1".Reading_Struct."32057",
                          DONE => "Modbus".Done,
                          BUSY => "Modbus".Busy,
                          ERROR => "Modbus".Error,
                          STATUS => "Modbus".Status);
   END_IF;
END_REGION

REGION Network 54: RD 32058
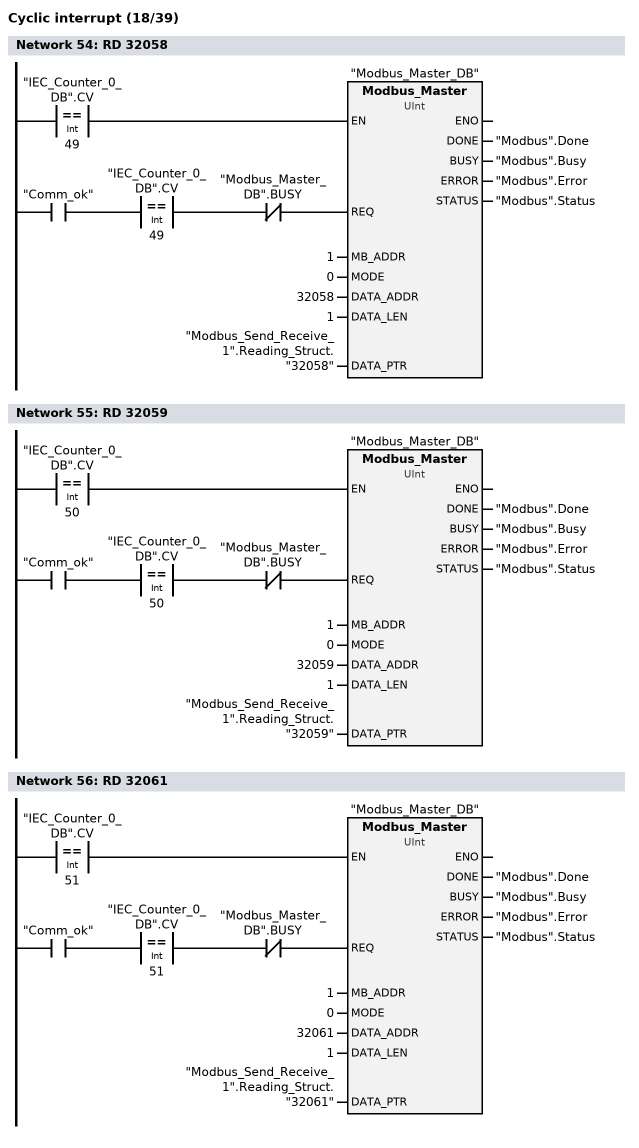
   RUNG wire#powerrail
      { S7_Templates := "SrcType := Int" } EQ_Contact(in1 := "IEC_Counter_0_DB".CV, in2 := 49)
      { S7_Templates := "[card := 0, word_type := UInt, dword_type := UDInt, byte_type := USInt, any_type := Variant]" } "Modbus_Master_DB".Modbus_Master(REQ := wire#w1, MB_ADDR := 1, MODE := 0, DATA_ADDR := 32058, DATA_LEN := 1, DATA_PTR := "Modbus_Send_Receive_1".Reading_Struct."32058", DONE => "Modbus".Done, BUSY => "Modbus".Busy, ERROR => "Modbus".Error, STATUS => "Modbus".Status)
   END_RUNG
   RUNG wire#powerrail
      Contact( "Comm_ok" )
      { S7_Templates := "SrcType := Int" } EQ_Contact(in1 := "IEC_Counter_0_DB".CV, in2 := 49)
      I_Contact( "Modbus_Master_DB".BUSY )
   END_RUNG wire#w1
   // the same network as SCL:
   IF "IEC_Counter_0_DB".CV = 49 THEN
       "Modbus_Master_DB"(REQ := "Comm_ok" AND ("IEC_Counter_0_DB".CV = 49) AND NOT "Modbus_Master_DB".BUSY,   // Modbus_Master
                          MB_ADDR := 1,
                          MODE := 0,
                          DATA_ADDR := 32058,
                          DATA_LEN := 1,
                          DATA_PTR := "Modbus_Send_Receive_1".Reading_Struct."32058",
                          DONE => "Modbus".Done,
                          BUSY => "Modbus".Busy,
                          ERROR => "Modbus".Error,
                          STATUS => "Modbus".Status);
   END_IF;
END_REGION

REGION Network 55: RD 32059
   RUNG wire#powerrail
      { S7_Templates := "SrcType := Int" } EQ_Contact(in1 := "IEC_Counter_0_DB".CV, in2 := 50)
      { S7_Templates := "[card := 0, word_type := UInt, dword_type := UDInt, byte_type := USInt, any_type := Variant]" } "Modbus_Master_DB".Modbus_Master(REQ := wire#w1, MB_ADDR := 1, MODE := 0, DATA_ADDR := 32059, DATA_LEN := 1, DATA_PTR := "Modbus_Send_Receive_1".Reading_Struct."32059", DONE => "Modbus".Done, BUSY => "Modbus".Busy, ERROR => "Modbus".Error, STATUS => "Modbus".Status)
   END_RUNG
   RUNG wire#powerrail
      Contact( "Comm_ok" )
      { S7_Templates := "SrcType := Int" } EQ_Contact(in1 := "IEC_Counter_0_DB".CV, in2 := 50)
      I_Contact( "Modbus_Master_DB".BUSY )
   END_RUNG wire#w1
   // the same network as SCL:
   IF "IEC_Counter_0_DB".CV = 50 THEN
       "Modbus_Master_DB"(REQ := "Comm_ok" AND ("IEC_Counter_0_DB".CV = 50) AND NOT "Modbus_Master_DB".BUSY,   // Modbus_Master
                          MB_ADDR := 1,
                          MODE := 0,
                          DATA_ADDR := 32059,
                          DATA_LEN := 1,
                          DATA_PTR := "Modbus_Send_Receive_1".Reading_Struct."32059",
                          DONE => "Modbus".Done,
                          BUSY => "Modbus".Busy,
                          ERROR => "Modbus".Error,
                          STATUS => "Modbus".Status);
   END_IF;
END_REGION

REGION Network 56: RD 32061
   RUNG wire#powerrail
      { S7_Templates := "SrcType := Int" } EQ_Contact(in1 := "IEC_Counter_0_DB".CV, in2 := 51)
      { S7_Templates := "[card := 0, word_type := UInt, dword_type := UDInt, byte_type := USInt, any_type := Variant]" } "Modbus_Master_DB".Modbus_Master(REQ := wire#w1, MB_ADDR := 1, MODE := 0, DATA_ADDR := 32061, DATA_LEN := 1, DATA_PTR := "Modbus_Send_Receive_1".Reading_Struct."32061", DONE => "Modbus".Done, BUSY => "Modbus".Busy, ERROR => "Modbus".Error, STATUS => "Modbus".Status)
   END_RUNG
   RUNG wire#powerrail
      Contact( "Comm_ok" )
      { S7_Templates := "SrcType := Int" } EQ_Contact(in1 := "IEC_Counter_0_DB".CV, in2 := 51)
      I_Contact( "Modbus_Master_DB".BUSY )
   END_RUNG wire#w1
   // the same network as SCL:
   IF "IEC_Counter_0_DB".CV = 51 THEN
       "Modbus_Master_DB"(REQ := "Comm_ok" AND ("IEC_Counter_0_DB".CV = 51) AND NOT "Modbus_Master_DB".BUSY,   // Modbus_Master
                          MB_ADDR := 1,
                          MODE := 0,
                          DATA_ADDR := 32061,
                          DATA_LEN := 1,
                          DATA_PTR := "Modbus_Send_Receive_1".Reading_Struct."32061",
                          DONE => "Modbus".Done,
                          BUSY => "Modbus".Busy,
                          ERROR => "Modbus".Error,
                          STATUS => "Modbus".Status);
   END_IF;
END_REGION

REGION Network 57: RD 32062
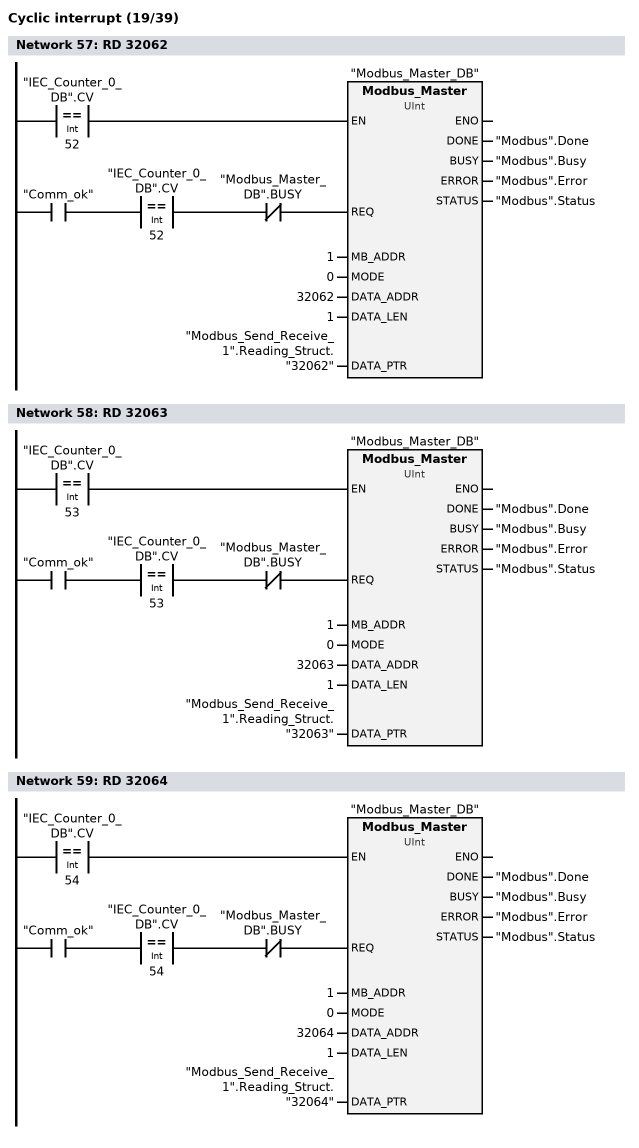
   RUNG wire#powerrail
      { S7_Templates := "SrcType := Int" } EQ_Contact(in1 := "IEC_Counter_0_DB".CV, in2 := 52)
      { S7_Templates := "[card := 0, word_type := UInt, dword_type := UDInt, byte_type := USInt, any_type := Variant]" } "Modbus_Master_DB".Modbus_Master(REQ := wire#w1, MB_ADDR := 1, MODE := 0, DATA_ADDR := 32062, DATA_LEN := 1, DATA_PTR := "Modbus_Send_Receive_1".Reading_Struct."32062", DONE => "Modbus".Done, BUSY => "Modbus".Busy, ERROR => "Modbus".Error, STATUS => "Modbus".Status)
   END_RUNG
   RUNG wire#powerrail
      Contact( "Comm_ok" )
      { S7_Templates := "SrcType := Int" } EQ_Contact(in1 := "IEC_Counter_0_DB".CV, in2 := 52)
      I_Contact( "Modbus_Master_DB".BUSY )
   END_RUNG wire#w1
   // the same network as SCL:
   IF "IEC_Counter_0_DB".CV = 52 THEN
       "Modbus_Master_DB"(REQ := "Comm_ok" AND ("IEC_Counter_0_DB".CV = 52) AND NOT "Modbus_Master_DB".BUSY,   // Modbus_Master
                          MB_ADDR := 1,
                          MODE := 0,
                          DATA_ADDR := 32062,
                          DATA_LEN := 1,
                          DATA_PTR := "Modbus_Send_Receive_1".Reading_Struct."32062",
                          DONE => "Modbus".Done,
                          BUSY => "Modbus".Busy,
                          ERROR => "Modbus".Error,
                          STATUS => "Modbus".Status);
   END_IF;
END_REGION

REGION Network 58: RD 32063
   RUNG wire#powerrail
      { S7_Templates := "SrcType := Int" } EQ_Contact(in1 := "IEC_Counter_0_DB".CV, in2 := 53)
      { S7_Templates := "[card := 0, word_type := UInt, dword_type := UDInt, byte_type := USInt, any_type := Variant]" } "Modbus_Master_DB".Modbus_Master(REQ := wire#w1, MB_ADDR := 1, MODE := 0, DATA_ADDR := 32063, DATA_LEN := 1, DATA_PTR := "Modbus_Send_Receive_1".Reading_Struct."32063", DONE => "Modbus".Done, BUSY => "Modbus".Busy, ERROR => "Modbus".Error, STATUS => "Modbus".Status)
   END_RUNG
   RUNG wire#powerrail
      Contact( "Comm_ok" )
      { S7_Templates := "SrcType := Int" } EQ_Contact(in1 := "IEC_Counter_0_DB".CV, in2 := 53)
      I_Contact( "Modbus_Master_DB".BUSY )
   END_RUNG wire#w1
   // the same network as SCL:
   IF "IEC_Counter_0_DB".CV = 53 THEN
       "Modbus_Master_DB"(REQ := "Comm_ok" AND ("IEC_Counter_0_DB".CV = 53) AND NOT "Modbus_Master_DB".BUSY,   // Modbus_Master
                          MB_ADDR := 1,
                          MODE := 0,
                          DATA_ADDR := 32063,
                          DATA_LEN := 1,
                          DATA_PTR := "Modbus_Send_Receive_1".Reading_Struct."32063",
                          DONE => "Modbus".Done,
                          BUSY => "Modbus".Busy,
                          ERROR => "Modbus".Error,
                          STATUS => "Modbus".Status);
   END_IF;
END_REGION

REGION Network 59: RD 32064
   RUNG wire#powerrail
      { S7_Templates := "SrcType := Int" } EQ_Contact(in1 := "IEC_Counter_0_DB".CV, in2 := 54)
      { S7_Templates := "[card := 0, word_type := UInt, dword_type := UDInt, byte_type := USInt, any_type := Variant]" } "Modbus_Master_DB".Modbus_Master(REQ := wire#w1, MB_ADDR := 1, MODE := 0, DATA_ADDR := 32064, DATA_LEN := 1, DATA_PTR := "Modbus_Send_Receive_1".Reading_Struct."32064", DONE => "Modbus".Done, BUSY => "Modbus".Busy, ERROR => "Modbus".Error, STATUS => "Modbus".Status)
   END_RUNG
   RUNG wire#powerrail
      Contact( "Comm_ok" )
      { S7_Templates := "SrcType := Int" } EQ_Contact(in1 := "IEC_Counter_0_DB".CV, in2 := 54)
      I_Contact( "Modbus_Master_DB".BUSY )
   END_RUNG wire#w1
   // the same network as SCL:
   IF "IEC_Counter_0_DB".CV = 54 THEN
       "Modbus_Master_DB"(REQ := "Comm_ok" AND ("IEC_Counter_0_DB".CV = 54) AND NOT "Modbus_Master_DB".BUSY,   // Modbus_Master
                          MB_ADDR := 1,
                          MODE := 0,
                          DATA_ADDR := 32064,
                          DATA_LEN := 1,
                          DATA_PTR := "Modbus_Send_Receive_1".Reading_Struct."32064",
                          DONE => "Modbus".Done,
                          BUSY => "Modbus".Busy,
                          ERROR => "Modbus".Error,
                          STATUS => "Modbus".Status);
   END_IF;
END_REGION

REGION Network 60: RD 32065
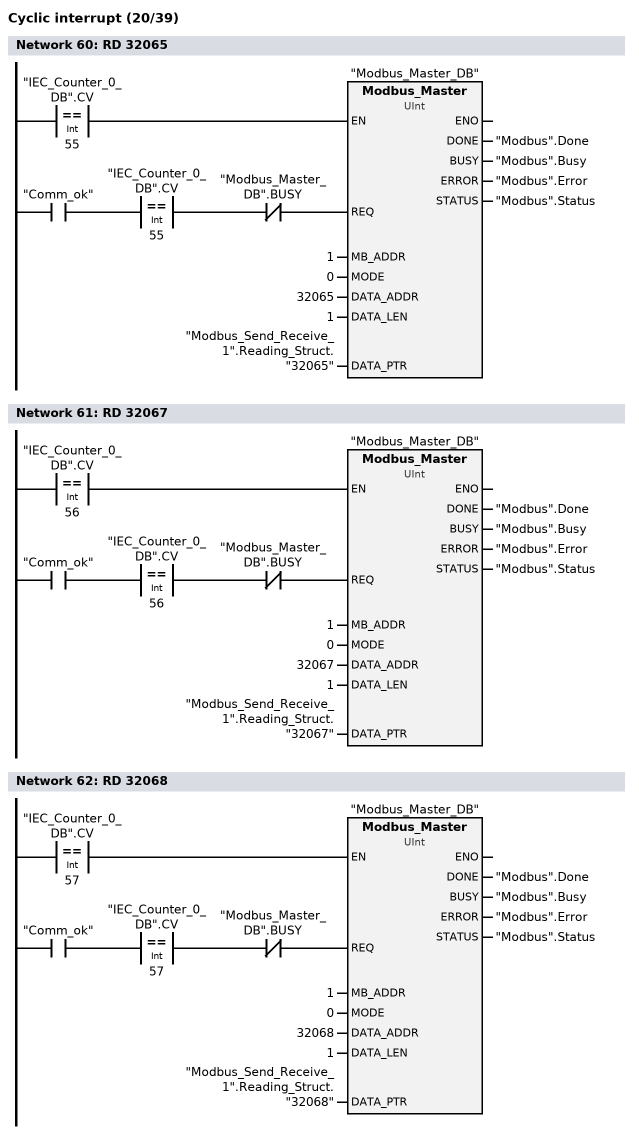
   RUNG wire#powerrail
      { S7_Templates := "SrcType := Int" } EQ_Contact(in1 := "IEC_Counter_0_DB".CV, in2 := 55)
      { S7_Templates := "[card := 0, word_type := UInt, dword_type := UDInt, byte_type := USInt, any_type := Variant]" } "Modbus_Master_DB".Modbus_Master(REQ := wire#w1, MB_ADDR := 1, MODE := 0, DATA_ADDR := 32065, DATA_LEN := 1, DATA_PTR := "Modbus_Send_Receive_1".Reading_Struct."32065", DONE => "Modbus".Done, BUSY => "Modbus".Busy, ERROR => "Modbus".Error, STATUS => "Modbus".Status)
   END_RUNG
   RUNG wire#powerrail
      Contact( "Comm_ok" )
      { S7_Templates := "SrcType := Int" } EQ_Contact(in1 := "IEC_Counter_0_DB".CV, in2 := 55)
      I_Contact( "Modbus_Master_DB".BUSY )
   END_RUNG wire#w1
   // the same network as SCL:
   IF "IEC_Counter_0_DB".CV = 55 THEN
       "Modbus_Master_DB"(REQ := "Comm_ok" AND ("IEC_Counter_0_DB".CV = 55) AND NOT "Modbus_Master_DB".BUSY,   // Modbus_Master
                          MB_ADDR := 1,
                          MODE := 0,
                          DATA_ADDR := 32065,
                          DATA_LEN := 1,
                          DATA_PTR := "Modbus_Send_Receive_1".Reading_Struct."32065",
                          DONE => "Modbus".Done,
                          BUSY => "Modbus".Busy,
                          ERROR => "Modbus".Error,
                          STATUS => "Modbus".Status);
   END_IF;
END_REGION

REGION Network 61: RD 32067
   RUNG wire#powerrail
      { S7_Templates := "SrcType := Int" } EQ_Contact(in1 := "IEC_Counter_0_DB".CV, in2 := 56)
      { S7_Templates := "[card := 0, word_type := UInt, dword_type := UDInt, byte_type := USInt, any_type := Variant]" } "Modbus_Master_DB".Modbus_Master(REQ := wire#w1, MB_ADDR := 1, MODE := 0, DATA_ADDR := 32067, DATA_LEN := 1, DATA_PTR := "Modbus_Send_Receive_1".Reading_Struct."32067", DONE => "Modbus".Done, BUSY => "Modbus".Busy, ERROR => "Modbus".Error, STATUS => "Modbus".Status)
   END_RUNG
   RUNG wire#powerrail
      Contact( "Comm_ok" )
      { S7_Templates := "SrcType := Int" } EQ_Contact(in1 := "IEC_Counter_0_DB".CV, in2 := 56)
      I_Contact( "Modbus_Master_DB".BUSY )
   END_RUNG wire#w1
   // the same network as SCL:
   IF "IEC_Counter_0_DB".CV = 56 THEN
       "Modbus_Master_DB"(REQ := "Comm_ok" AND ("IEC_Counter_0_DB".CV = 56) AND NOT "Modbus_Master_DB".BUSY,   // Modbus_Master
                          MB_ADDR := 1,
                          MODE := 0,
                          DATA_ADDR := 32067,
                          DATA_LEN := 1,
                          DATA_PTR := "Modbus_Send_Receive_1".Reading_Struct."32067",
                          DONE => "Modbus".Done,
                          BUSY => "Modbus".Busy,
                          ERROR => "Modbus".Error,
                          STATUS => "Modbus".Status);
   END_IF;
END_REGION

REGION Network 62: RD 32068
   RUNG wire#powerrail
      { S7_Templates := "SrcType := Int" } EQ_Contact(in1 := "IEC_Counter_0_DB".CV, in2 := 57)
      { S7_Templates := "[card := 0, word_type := UInt, dword_type := UDInt, byte_type := USInt, any_type := Variant]" } "Modbus_Master_DB".Modbus_Master(REQ := wire#w1, MB_ADDR := 1, MODE := 0, DATA_ADDR := 32068, DATA_LEN := 1, DATA_PTR := "Modbus_Send_Receive_1".Reading_Struct."32068", DONE => "Modbus".Done, BUSY => "Modbus".Busy, ERROR => "Modbus".Error, STATUS => "Modbus".Status)
   END_RUNG
   RUNG wire#powerrail
      Contact( "Comm_ok" )
      { S7_Templates := "SrcType := Int" } EQ_Contact(in1 := "IEC_Counter_0_DB".CV, in2 := 57)
      I_Contact( "Modbus_Master_DB".BUSY )
   END_RUNG wire#w1
   // the same network as SCL:
   IF "IEC_Counter_0_DB".CV = 57 THEN
       "Modbus_Master_DB"(REQ := "Comm_ok" AND ("IEC_Counter_0_DB".CV = 57) AND NOT "Modbus_Master_DB".BUSY,   // Modbus_Master
                          MB_ADDR := 1,
                          MODE := 0,
                          DATA_ADDR := 32068,
                          DATA_LEN := 1,
                          DATA_PTR := "Modbus_Send_Receive_1".Reading_Struct."32068",
                          DONE => "Modbus".Done,
                          BUSY => "Modbus".Busy,
                          ERROR => "Modbus".Error,
                          STATUS => "Modbus".Status);
   END_IF;
END_REGION

REGION Network 63: RD 32069
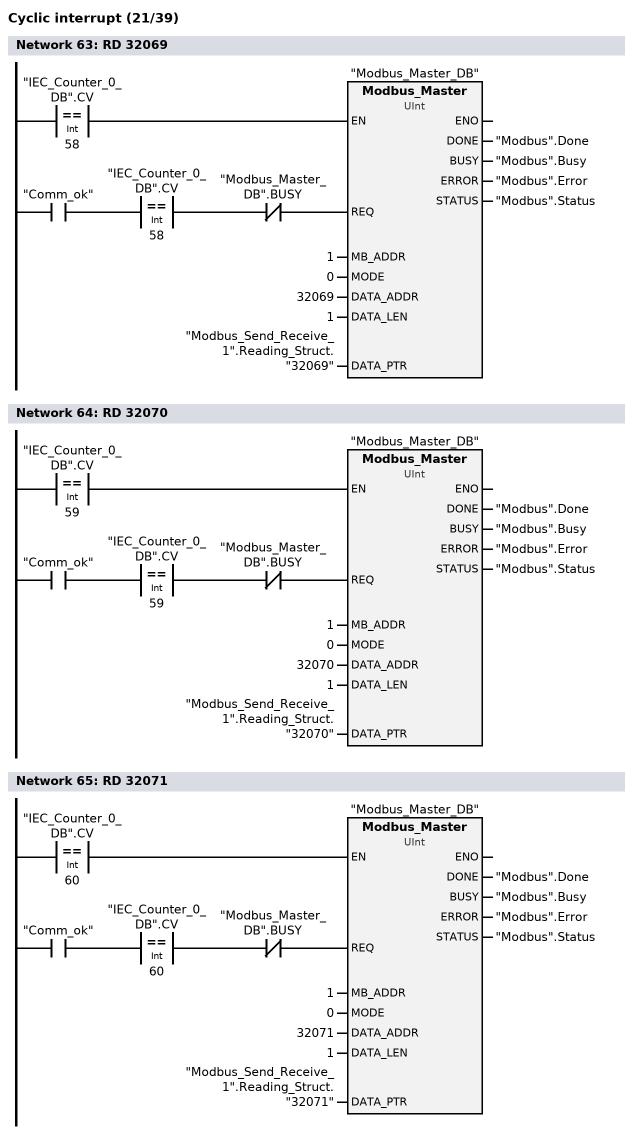
   RUNG wire#powerrail
      { S7_Templates := "SrcType := Int" } EQ_Contact(in1 := "IEC_Counter_0_DB".CV, in2 := 58)
      { S7_Templates := "[card := 0, word_type := UInt, dword_type := UDInt, byte_type := USInt, any_type := Variant]" } "Modbus_Master_DB".Modbus_Master(REQ := wire#w1, MB_ADDR := 1, MODE := 0, DATA_ADDR := 32069, DATA_LEN := 1, DATA_PTR := "Modbus_Send_Receive_1".Reading_Struct."32069", DONE => "Modbus".Done, BUSY => "Modbus".Busy, ERROR => "Modbus".Error, STATUS => "Modbus".Status)
   END_RUNG
   RUNG wire#powerrail
      Contact( "Comm_ok" )
      { S7_Templates := "SrcType := Int" } EQ_Contact(in1 := "IEC_Counter_0_DB".CV, in2 := 58)
      I_Contact( "Modbus_Master_DB".BUSY )
   END_RUNG wire#w1
   // the same network as SCL:
   IF "IEC_Counter_0_DB".CV = 58 THEN
       "Modbus_Master_DB"(REQ := "Comm_ok" AND ("IEC_Counter_0_DB".CV = 58) AND NOT "Modbus_Master_DB".BUSY,   // Modbus_Master
                          MB_ADDR := 1,
                          MODE := 0,
                          DATA_ADDR := 32069,
                          DATA_LEN := 1,
                          DATA_PTR := "Modbus_Send_Receive_1".Reading_Struct."32069",
                          DONE => "Modbus".Done,
                          BUSY => "Modbus".Busy,
                          ERROR => "Modbus".Error,
                          STATUS => "Modbus".Status);
   END_IF;
END_REGION

REGION Network 64: RD 32070
   RUNG wire#powerrail
      { S7_Templates := "SrcType := Int" } EQ_Contact(in1 := "IEC_Counter_0_DB".CV, in2 := 59)
      { S7_Templates := "[card := 0, word_type := UInt, dword_type := UDInt, byte_type := USInt, any_type := Variant]" } "Modbus_Master_DB".Modbus_Master(REQ := wire#w1, MB_ADDR := 1, MODE := 0, DATA_ADDR := 32070, DATA_LEN := 1, DATA_PTR := "Modbus_Send_Receive_1".Reading_Struct."32070", DONE => "Modbus".Done, BUSY => "Modbus".Busy, ERROR => "Modbus".Error, STATUS => "Modbus".Status)
   END_RUNG
   RUNG wire#powerrail
      Contact( "Comm_ok" )
      { S7_Templates := "SrcType := Int" } EQ_Contact(in1 := "IEC_Counter_0_DB".CV, in2 := 59)
      I_Contact( "Modbus_Master_DB".BUSY )
   END_RUNG wire#w1
   // the same network as SCL:
   IF "IEC_Counter_0_DB".CV = 59 THEN
       "Modbus_Master_DB"(REQ := "Comm_ok" AND ("IEC_Counter_0_DB".CV = 59) AND NOT "Modbus_Master_DB".BUSY,   // Modbus_Master
                          MB_ADDR := 1,
                          MODE := 0,
                          DATA_ADDR := 32070,
                          DATA_LEN := 1,
                          DATA_PTR := "Modbus_Send_Receive_1".Reading_Struct."32070",
                          DONE => "Modbus".Done,
                          BUSY => "Modbus".Busy,
                          ERROR => "Modbus".Error,
                          STATUS => "Modbus".Status);
   END_IF;
END_REGION

REGION Network 65: RD 32071
   RUNG wire#powerrail
      { S7_Templates := "SrcType := Int" } EQ_Contact(in1 := "IEC_Counter_0_DB".CV, in2 := 60)
      { S7_Templates := "[card := 0, word_type := UInt, dword_type := UDInt, byte_type := USInt, any_type := Variant]" } "Modbus_Master_DB".Modbus_Master(REQ := wire#w1, MB_ADDR := 1, MODE := 0, DATA_ADDR := 32071, DATA_LEN := 1, DATA_PTR := "Modbus_Send_Receive_1".Reading_Struct."32071", DONE => "Modbus".Done, BUSY => "Modbus".Busy, ERROR => "Modbus".Error, STATUS => "Modbus".Status)
   END_RUNG
   RUNG wire#powerrail
      Contact( "Comm_ok" )
      { S7_Templates := "SrcType := Int" } EQ_Contact(in1 := "IEC_Counter_0_DB".CV, in2 := 60)
      I_Contact( "Modbus_Master_DB".BUSY )
   END_RUNG wire#w1
   // the same network as SCL:
   IF "IEC_Counter_0_DB".CV = 60 THEN
       "Modbus_Master_DB"(REQ := "Comm_ok" AND ("IEC_Counter_0_DB".CV = 60) AND NOT "Modbus_Master_DB".BUSY,   // Modbus_Master
                          MB_ADDR := 1,
                          MODE := 0,
                          DATA_ADDR := 32071,
                          DATA_LEN := 1,
                          DATA_PTR := "Modbus_Send_Receive_1".Reading_Struct."32071",
                          DONE => "Modbus".Done,
                          BUSY => "Modbus".Busy,
                          ERROR => "Modbus".Error,
                          STATUS => "Modbus".Status);
   END_IF;
END_REGION

REGION Network 66: RD 32073
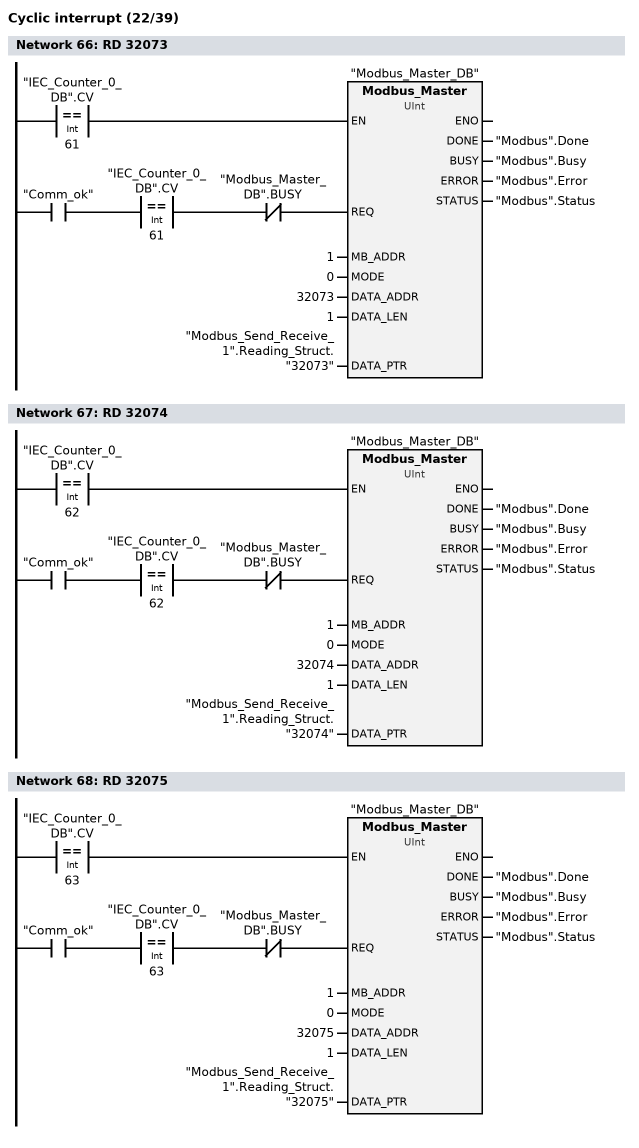
   RUNG wire#powerrail
      { S7_Templates := "SrcType := Int" } EQ_Contact(in1 := "IEC_Counter_0_DB".CV, in2 := 61)
      { S7_Templates := "[card := 0, word_type := UInt, dword_type := UDInt, byte_type := USInt, any_type := Variant]" } "Modbus_Master_DB".Modbus_Master(REQ := wire#w1, MB_ADDR := 1, MODE := 0, DATA_ADDR := 32073, DATA_LEN := 1, DATA_PTR := "Modbus_Send_Receive_1".Reading_Struct."32073", DONE => "Modbus".Done, BUSY => "Modbus".Busy, ERROR => "Modbus".Error, STATUS => "Modbus".Status)
   END_RUNG
   RUNG wire#powerrail
      Contact( "Comm_ok" )
      { S7_Templates := "SrcType := Int" } EQ_Contact(in1 := "IEC_Counter_0_DB".CV, in2 := 61)
      I_Contact( "Modbus_Master_DB".BUSY )
   END_RUNG wire#w1
   // the same network as SCL:
   IF "IEC_Counter_0_DB".CV = 61 THEN
       "Modbus_Master_DB"(REQ := "Comm_ok" AND ("IEC_Counter_0_DB".CV = 61) AND NOT "Modbus_Master_DB".BUSY,   // Modbus_Master
                          MB_ADDR := 1,
                          MODE := 0,
                          DATA_ADDR := 32073,
                          DATA_LEN := 1,
                          DATA_PTR := "Modbus_Send_Receive_1".Reading_Struct."32073",
                          DONE => "Modbus".Done,
                          BUSY => "Modbus".Busy,
                          ERROR => "Modbus".Error,
                          STATUS => "Modbus".Status);
   END_IF;
END_REGION

REGION Network 67: RD 32074
   RUNG wire#powerrail
      { S7_Templates := "SrcType := Int" } EQ_Contact(in1 := "IEC_Counter_0_DB".CV, in2 := 62)
      { S7_Templates := "[card := 0, word_type := UInt, dword_type := UDInt, byte_type := USInt, any_type := Variant]" } "Modbus_Master_DB".Modbus_Master(REQ := wire#w1, MB_ADDR := 1, MODE := 0, DATA_ADDR := 32074, DATA_LEN := 1, DATA_PTR := "Modbus_Send_Receive_1".Reading_Struct."32074", DONE => "Modbus".Done, BUSY => "Modbus".Busy, ERROR => "Modbus".Error, STATUS => "Modbus".Status)
   END_RUNG
   RUNG wire#powerrail
      Contact( "Comm_ok" )
      { S7_Templates := "SrcType := Int" } EQ_Contact(in1 := "IEC_Counter_0_DB".CV, in2 := 62)
      I_Contact( "Modbus_Master_DB".BUSY )
   END_RUNG wire#w1
   // the same network as SCL:
   IF "IEC_Counter_0_DB".CV = 62 THEN
       "Modbus_Master_DB"(REQ := "Comm_ok" AND ("IEC_Counter_0_DB".CV = 62) AND NOT "Modbus_Master_DB".BUSY,   // Modbus_Master
                          MB_ADDR := 1,
                          MODE := 0,
                          DATA_ADDR := 32074,
                          DATA_LEN := 1,
                          DATA_PTR := "Modbus_Send_Receive_1".Reading_Struct."32074",
                          DONE => "Modbus".Done,
                          BUSY => "Modbus".Busy,
                          ERROR => "Modbus".Error,
                          STATUS => "Modbus".Status);
   END_IF;
END_REGION

REGION Network 68: RD 32075
   RUNG wire#powerrail
      { S7_Templates := "SrcType := Int" } EQ_Contact(in1 := "IEC_Counter_0_DB".CV, in2 := 63)
      { S7_Templates := "[card := 0, word_type := UInt, dword_type := UDInt, byte_type := USInt, any_type := Variant]" } "Modbus_Master_DB".Modbus_Master(REQ := wire#w1, MB_ADDR := 1, MODE := 0, DATA_ADDR := 32075, DATA_LEN := 1, DATA_PTR := "Modbus_Send_Receive_1".Reading_Struct."32075", DONE => "Modbus".Done, BUSY => "Modbus".Busy, ERROR => "Modbus".Error, STATUS => "Modbus".Status)
   END_RUNG
   RUNG wire#powerrail
      Contact( "Comm_ok" )
      { S7_Templates := "SrcType := Int" } EQ_Contact(in1 := "IEC_Counter_0_DB".CV, in2 := 63)
      I_Contact( "Modbus_Master_DB".BUSY )
   END_RUNG wire#w1
   // the same network as SCL:
   IF "IEC_Counter_0_DB".CV = 63 THEN
       "Modbus_Master_DB"(REQ := "Comm_ok" AND ("IEC_Counter_0_DB".CV = 63) AND NOT "Modbus_Master_DB".BUSY,   // Modbus_Master
                          MB_ADDR := 1,
                          MODE := 0,
                          DATA_ADDR := 32075,
                          DATA_LEN := 1,
                          DATA_PTR := "Modbus_Send_Receive_1".Reading_Struct."32075",
                          DONE => "Modbus".Done,
                          BUSY => "Modbus".Busy,
                          ERROR => "Modbus".Error,
                          STATUS => "Modbus".Status);
   END_IF;
END_REGION

REGION Network 69: RD 32076
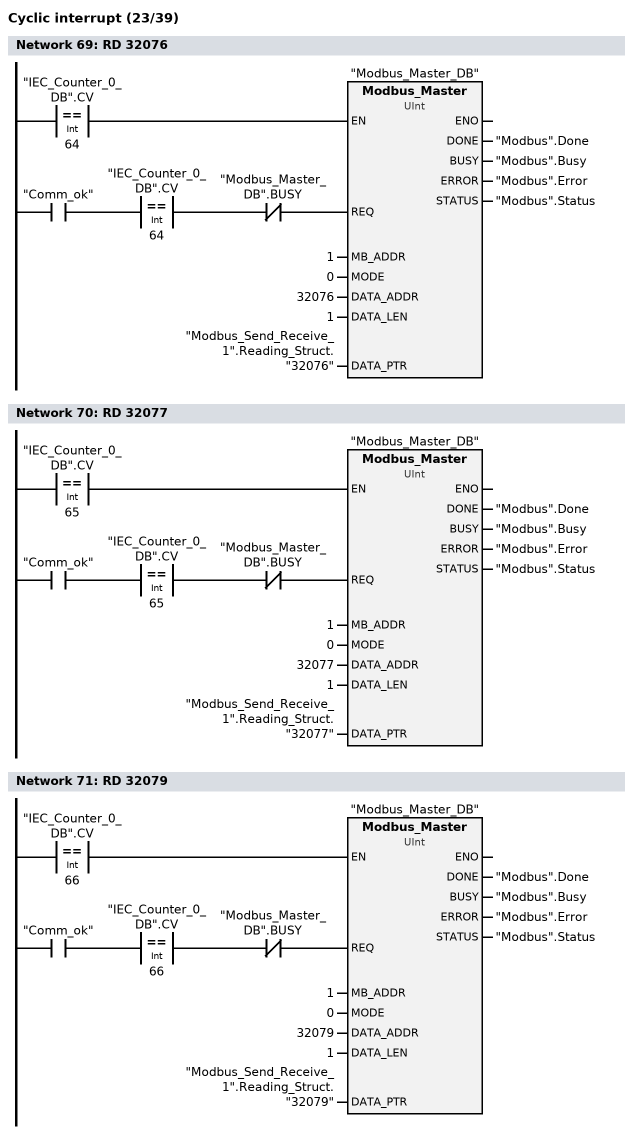
   RUNG wire#powerrail
      { S7_Templates := "SrcType := Int" } EQ_Contact(in1 := "IEC_Counter_0_DB".CV, in2 := 64)
      { S7_Templates := "[card := 0, word_type := UInt, dword_type := UDInt, byte_type := USInt, any_type := Variant]" } "Modbus_Master_DB".Modbus_Master(REQ := wire#w1, MB_ADDR := 1, MODE := 0, DATA_ADDR := 32076, DATA_LEN := 1, DATA_PTR := "Modbus_Send_Receive_1".Reading_Struct."32076", DONE => "Modbus".Done, BUSY => "Modbus".Busy, ERROR => "Modbus".Error, STATUS => "Modbus".Status)
   END_RUNG
   RUNG wire#powerrail
      Contact( "Comm_ok" )
      { S7_Templates := "SrcType := Int" } EQ_Contact(in1 := "IEC_Counter_0_DB".CV, in2 := 64)
      I_Contact( "Modbus_Master_DB".BUSY )
   END_RUNG wire#w1
   // the same network as SCL:
   IF "IEC_Counter_0_DB".CV = 64 THEN
       "Modbus_Master_DB"(REQ := "Comm_ok" AND ("IEC_Counter_0_DB".CV = 64) AND NOT "Modbus_Master_DB".BUSY,   // Modbus_Master
                          MB_ADDR := 1,
                          MODE := 0,
                          DATA_ADDR := 32076,
                          DATA_LEN := 1,
                          DATA_PTR := "Modbus_Send_Receive_1".Reading_Struct."32076",
                          DONE => "Modbus".Done,
                          BUSY => "Modbus".Busy,
                          ERROR => "Modbus".Error,
                          STATUS => "Modbus".Status);
   END_IF;
END_REGION

REGION Network 70: RD 32077
   RUNG wire#powerrail
      { S7_Templates := "SrcType := Int" } EQ_Contact(in1 := "IEC_Counter_0_DB".CV, in2 := 65)
      { S7_Templates := "[card := 0, word_type := UInt, dword_type := UDInt, byte_type := USInt, any_type := Variant]" } "Modbus_Master_DB".Modbus_Master(REQ := wire#w1, MB_ADDR := 1, MODE := 0, DATA_ADDR := 32077, DATA_LEN := 1, DATA_PTR := "Modbus_Send_Receive_1".Reading_Struct."32077", DONE => "Modbus".Done, BUSY => "Modbus".Busy, ERROR => "Modbus".Error, STATUS => "Modbus".Status)
   END_RUNG
   RUNG wire#powerrail
      Contact( "Comm_ok" )
      { S7_Templates := "SrcType := Int" } EQ_Contact(in1 := "IEC_Counter_0_DB".CV, in2 := 65)
      I_Contact( "Modbus_Master_DB".BUSY )
   END_RUNG wire#w1
   // the same network as SCL:
   IF "IEC_Counter_0_DB".CV = 65 THEN
       "Modbus_Master_DB"(REQ := "Comm_ok" AND ("IEC_Counter_0_DB".CV = 65) AND NOT "Modbus_Master_DB".BUSY,   // Modbus_Master
                          MB_ADDR := 1,
                          MODE := 0,
                          DATA_ADDR := 32077,
                          DATA_LEN := 1,
                          DATA_PTR := "Modbus_Send_Receive_1".Reading_Struct."32077",
                          DONE => "Modbus".Done,
                          BUSY => "Modbus".Busy,
                          ERROR => "Modbus".Error,
                          STATUS => "Modbus".Status);
   END_IF;
END_REGION

